LIN {X 0,Y 305.497,Z 546.552,A -85,B 0,C 180,E1 -15897.566,E2 -15897.566} C_VEL
LIN {X 0,Y 308.122,Z 558.584,A -85,B 0,C 180,E1 -15901.379,E2 -15901.379} C_VEL
LIN {X 0,Y 309.792,Z 567.618,A -85,B 0,C 180,E1 -15904.104,E2 -15904.104} C_VEL
LIN {X 0,Y 309.747,Z 569.897,A -85,B 0,C 180,E1 -15904.748,E2 -15904.748} C_VEL
LIN {X 0,Y 315.852,Z 610.316,A -85,B 0,C 180,E1 -15906.253,E2 -15906.253} C_VEL
LIN {X 0,Y 314.086,Z 678.463,A -85,B 0,C 180,E1 -15907.943,E2 -15907.943} C_VEL
LIN {X 0,Y 313.22,Z 691.999,A -85,B 0,C 180,E1 -15908.528,E2 -15908.528} C_VEL
LIN {X 0,Y 312.136,Z 704.365,A -85,B 0,C 180,E1 -15909.314,E2 -15909.314} C_VEL
LIN {X 0,Y 310.892,Z 716.286,A -85,B 0,C 180,E1 -15910.349,E2 -15910.349} C_VEL
LIN {X 0,Y 309.544,Z 727.77,A -85,B 0,C 180,E1 -15911.636,E2 -15911.636} C_VEL
LIN {X 0,Y 308.303,Z 737.547,A -85,B 0,C 180,E1 -15913.006,E2 -15913.006} C_VEL
LIN {X 0,Y 307.077,Z 747.457,A -85,B 0,C 180,E1 -15914.738,E2 -15914.738} C_VEL
LIN {X 0,Y 305.804,Z 756.501,A -85,B 0,C 180,E1 -15916.712,E2 -15916.712} C_VEL
LIN {X 0,Y 304.877,Z 763.765,A -85,B 0,C 180,E1 -15918.698,E2 -15918.698} C_VEL
LIN {X 0,Y 304.247,Z 769.534,A -85,B 0,C 180,E1 -15920.693,E2 -15920.693} C_VEL
LIN {X 0,Y 303.857,Z 774.057,A -85,B 0,C 180,E1 -15922.69,E2 -15922.69} C_VEL
LIN {X 0,Y 303.669,Z 777.467,A -85,B 0,C 180,E1 -15924.686,E2 -15924.686} C_VEL
LIN {X 0,Y 303.642,Z 779.152,A -85,B 0,C 180,E1 -15926.016,E2 -15926.016} C_VEL
LIN {X 0,Y 303.61,Z 780.42,A -85,B 0,C 180,E1 -15927.345,E2 -15927.345} C_VEL
LIN {X 0,Y 303.577,Z 781.275,A -85,B 0,C 180,E1 -15928.672,E2 -15928.672} C_VEL
LIN {X 0,Y 303.605,Z 781.68,A -85,B 0,C 180,E1 -15929.998,E2 -15929.998} C_VEL
LIN {X 0,Y 303.567,Z 781.681,A -85,B 0,C 180,E1 -15931.325,E2 -15931.325} C_VEL
LIN {X 0,Y 303.604,Z 781.289,A -85,B 0,C 180,E1 -15932.652,E2 -15932.652} C_VEL
LIN {X 0,Y 303.599,Z 780.496,A -85,B 0,C 180,E1 -15933.98,E2 -15933.98} C_VEL
LIN {X 0,Y 303.626,Z 778.989,A -85,B 0,C 180,E1 -15935.543,E2 -15935.543} C_VEL
LIN {X 0,Y 303.993,Z 775.521,A -85,B 0,C 180,E1 -15937.971,E2 -15937.971} C_VEL
LIN {X 0,Y 304.505,Z 771.506,A -85,B 0,C 180,E1 -15939.966,E2 -15939.966} C_VEL
LIN {X 0,Y 305.464,Z 765.357,A -85,B 0,C 180,E1 -15942.286,E2 -15942.286} C_VEL
LIN {X 0,Y 306.731,Z 758.652,A -85,B 0,C 180,E1 -15944.257,E2 -15944.257} C_VEL
LIN {X 0,Y 308.205,Z 750.629,A -85,B 0,C 180,E1 -15946.157,E2 -15946.157} C_VEL
LIN {X 0,Y 309.648,Z 741.904,A -85,B 0,C 180,E1 -15947.84,E2 -15947.84} C_VEL
LIN {X 0,Y 311.396,Z 731.495,A -85,B 0,C 180,E1 -15949.443,E2 -15949.443} C_VEL
LIN {X 0,Y 313.245,Z 719.826,A -85,B 0,C 180,E1 -15950.863,E2 -15950.863} C_VEL
LIN {X 0,Y 314.876,Z 708.285,A -85,B 0,C 180,E1 -15951.952,E2 -15951.952} C_VEL
LIN {X 0,Y 316.109,Z 696.459,A -85,B 0,C 180,E1 -15952.808,E2 -15952.808} C_VEL
LIN {X 0,Y 317.302,Z 683.01,A -85,B 0,C 180,E1 -15953.494,E2 -15953.494} C_VEL
LIN {X 0,Y 318.066,Z 670,A -85,B 0,C 180,E1 -15953.9,E2 -15953.9} C_VEL
LIN {X 0,Y 319.853,Z 610.651,A -85,B 0,C 180,E1 -15955.385,E2 -15955.385} C_VEL
LIN {X 0,Y 316.871,Z 591.359,A -85,B 0,C 180,E1 -15956.251,E2 -15956.251} C_VEL
LIN {X 0,Y 313.731,Z 576.118,A -85,B 0,C 180,E1 -15957.04,E2 -15957.04} C_VEL
LIN {X 0,Y 310.518,Z 568.505,A -85,B 0,C 180,E1 -15957.655,E2 -15957.655} C_VEL
LIN {X 0,Y 309.018,Z 560.982,A -85,B 0,C 180,E1 -15960.203,E2 -15960.203} C_VEL
LIN {X 0,Y 306.966,Z 552.375,A -85,B 0,C 180,E1 -15963.329,E2 -15963.329} C_VEL
LIN {X 0,Y 305.5,Z 546.432,A -85,B 0,C 180,E1 -15965.712,E2 -15965.712} C_VEL
LIN {X 0,Y 305.488,Z 546.436,A -85,B 0,C 180,E1 -15968.537,E2 -15968.537} C_VEL
LIN {X 0,Y 305.483,Z 546.436,A -85,B 0,C 180,E1 -15972.591,E2 -15972.591} C_VEL
LIN {X 0,Y 305.482,Z 546.432,A -85,B 0,C 180,E1 -15977.405,E2 -15977.405} C_VEL
LIN {X 0,Y 305.501,Z 546.43,A -85,B 0,C 180,E1 -15981.601,E2 -15981.601} C_VEL
LIN {X 0,Y 305.455,Z 546.436,A -85,B 0,C 180,E1 -15984.885,E2 -15984.885} C_VEL
LIN {X 0,Y 305.444,Z 546.435,A -85,B 0,C 180,E1 -15988.353,E2 -15988.353} C_VEL
LIN {X 0,Y 305.512,Z 546.43,A -85,B 0,C 180,E1 -15991.112,E2 -15991.112} C_VEL
LIN {X 0,Y 305.562,Z 546.423,A -85,B 0,C 180,E1 -15994.086,E2 -15994.086} C_VEL
LIN {X 0,Y 305.491,Z 546.431,A -85,B 0,C 180,E1 -15998.401,E2 -15998.401} C_VEL
LIN {X 0,Y 305.58,Z 546.413,A -85,B 0,C 180,E1 -16001.216,E2 -16001.216} C_VEL
LIN {X 0,Y 305.638,Z 546.409,A -85,B 0,C 180,E1 -16005.348,E2 -16005.348} C_VEL
LIN {X 0,Y 305.63,Z 546.412,A -85,B 0,C 180,E1 -16009.399,E2 -16009.399} C_VEL
LIN {X 0,Y 305.802,Z 546.386,A -85,B 0,C 180,E1 -16012.073,E2 -16012.073} C_VEL
LIN {X 0,Y 305.68,Z 546.405,A -85,B 0,C 180,E1 -16014.723,E2 -16014.723} C_VEL
LIN {X 0,Y 305.95,Z 546.368,A -85,B 0,C 180,E1 -16018.683,E2 -16018.683} C_VEL
LIN {X 0,Y 305.95,Z 546.372,A -85,B 0,C 180,E1 -16021.316,E2 -16021.316} C_VEL
LIN {X 0,Y 305.682,Z 546.405,A -85,B 0,C 180,E1 -16025.276,E2 -16025.276} C_VEL
LIN {X 0,Y 305.802,Z 546.392,A -85,B 0,C 180,E1 -16027.925,E2 -16027.925} C_VEL
LIN {X 0,Y 305.595,Z 546.418,A -85,B 0,C 180,E1 -16031.945,E2 -16031.945} C_VEL
LIN {X 0,Y 305.626,Z 546.419,A -85,B 0,C 180,E1 -16035.035,E2 -16035.035} C_VEL
LIN {X 0,Y 305.596,Z 546.587,A -85,B 0,C 180,E1 -16038.607,E2 -16038.607} C_VEL
LIN {X 0,Y 307.529,Z 554.976,A -85,B 0,C 180,E1 -16042.064,E2 -16042.064} C_VEL
LIN {X 0,Y 316.004,Z 572.925,A -85,B 0,C 180,E1 -16043.598,E2 -16043.598} C_VEL
LIN {X 0,Y 319.551,Z 581.78,A -85,B 0,C 180,E1 -16044.238,E2 -16044.238} C_VEL
LIN {X 0,Y 320.605,Z 586.987,A -85,B 0,C 180,E1 -16044.497,E2 -16044.497} C_VEL
LIN {X 0,Y 318.005,Z 661.781,A -85,B 0,C 180,E1 -16046.382,E2 -16046.382} C_VEL
LIN {X 0,Y 317.129,Z 675.045,A -85,B 0,C 180,E1 -16046.96,E2 -16046.96} C_VEL
LIN {X 0,Y 316.022,Z 687.675,A -85,B 0,C 180,E1 -16047.771,E2 -16047.771} C_VEL
LIN {X 0,Y 314.756,Z 698.402,A -85,B 0,C 180,E1 -16048.689,E2 -16048.689} C_VEL
LIN {X 0,Y 313.17,Z 709.886,A -85,B 0,C 180,E1 -16049.954,E2 -16049.954} C_VEL
LIN {X 0,Y 311.449,Z 720.68,A -85,B 0,C 180,E1 -16051.454,E2 -16051.454} C_VEL
LIN {X 0,Y 309.689,Z 730.59,A -85,B 0,C 180,E1 -16053.194,E2 -16053.194} C_VEL
LIN {X 0,Y 308.019,Z 739.585,A -85,B 0,C 180,E1 -16055.182,E2 -16055.182} C_VEL
LIN {X 0,Y 306.727,Z 746.339,A -85,B 0,C 180,E1 -16057.049,E2 -16057.049} C_VEL
LIN {X 0,Y 305.478,Z 752.794,A -85,B 0,C 180,E1 -16059.333,E2 -16059.333} C_VEL
LIN {X 0,Y 304.787,Z 756.885,A -85,B 0,C 180,E1 -16061.202,E2 -16061.202} C_VEL
LIN {X 0,Y 304.193,Z 760.192,A -85,B 0,C 180,E1 -16063.191,E2 -16063.191} C_VEL
LIN {X 0,Y 303.966,Z 761.501,A -85,B 0,C 180,E1 -16064.216,E2 -16064.216} C_VEL
LIN {X 0,Y 303.625,Z 763.205,A -85,B 0,C 180,E1 -16066.023,E2 -16066.023} C_VEL
LIN {X 0,Y 303.417,Z 764.115,A -85,B 0,C 180,E1 -16067.833,E2 -16067.833} C_VEL
LIN {X 0,Y 303.29,Z 764.261,A -85,B 0,C 180,E1 -16069.879,E2 -16069.879} C_VEL
LIN {X 0,Y 303.332,Z 763.417,A -85,B 0,C 180,E1 -16071.975,E2 -16071.975} C_VEL
LIN {X 0,Y 303.671,Z 760.861,A -85,B 0,C 180,E1 -16074.652,E2 -16074.652} C_VEL
LIN {X 0,Y 304.083,Z 756.872,A -85,B 0,C 180,E1 -16077.134,E2 -16077.134} C_VEL
LIN {X 0,Y 304.716,Z 751.498,A -85,B 0,C 180,E1 -16079.511,E2 -16079.511} C_VEL
LIN {X 0,Y 305.463,Z 745.633,A -85,B 0,C 180,E1 -16081.486,E2 -16081.486} C_VEL
LIN {X 0,Y 306.437,Z 738.38,A -85,B 0,C 180,E1 -16083.436,E2 -16083.436} C_VEL
LIN {X 0,Y 307.701,Z 729.421,A -85,B 0,C 180,E1 -16085.367,E2 -16085.367} C_VEL
LIN {X 0,Y 308.945,Z 719.517,A -85,B 0,C 180,E1 -16087.075,E2 -16087.075} C_VEL
LIN {X 0,Y 310.344,Z 708.853,A -85,B 0,C 180,E1 -16088.538,E2 -16088.538} C_VEL
LIN {X 0,Y 311.485,Z 698.278,A -85,B 0,C 180,E1 -16089.704,E2 -16089.704} C_VEL
LIN {X 0,Y 312.546,Z 687.241,A -85,B 0,C 180,E1 -16090.664,E2 -16090.664} C_VEL
LIN {X 0,Y 313.439,Z 674.541,A -85,B 0,C 180,E1 -16091.488,E2 -16091.488} C_VEL
LIN {X 0,Y 314.186,Z 660.798,A -85,B 0,C 180,E1 -16092.089,E2 -16092.089} C_VEL
LIN {X 0,Y 316.226,Z 584.792,A -85,B 0,C 180,E1 -16093.966,E2 -16093.966} C_VEL
LIN {X 0,Y 313.519,Z 571.685,A -85,B 0,C 180,E1 -16094.502,E2 -16094.502} C_VEL
LIN {X 0,Y 307.021,Z 553.372,A -85,B 0,C 180,E1 -16095.503,E2 -16095.503} C_VEL
LIN {X 0,Y 305.625,Z 546.415,A -85,B 0,C 180,E1 -16097.974,E2 -16097.974} C_VEL
LIN {X 0,Y 305.799,Z 546.392,A -85,B 0,C 180,E1 -16102.076,E2 -16102.076} C_VEL
LIN {X 0,Y 305.684,Z 546.411,A -85,B 0,C 180,E1 -16104.725,E2 -16104.725} C_VEL
LIN {X 0,Y 305.954,Z 546.375,A -85,B 0,C 180,E1 -16108.686,E2 -16108.686} C_VEL
LIN {X 0,Y 305.955,Z 546.373,A -85,B 0,C 180,E1 -16111.318,E2 -16111.318} C_VEL
LIN {X 0,Y 305.844,Z 546.385,A -85,B 0,C 180,E1 -16116.599,E2 -16116.599} C_VEL
LIN {X 0,Y 305.734,Z 546.402,A -85,B 0,C 180,E1 -16119.262,E2 -16119.262} C_VEL
LIN {X 0,Y 305.588,Z 546.418,A -85,B 0,C 180,E1 -16123.298,E2 -16123.298} C_VEL
LIN {X 0,Y 305.593,Z 546.416,A -85,B 0,C 180,E1 -16126.022,E2 -16126.022} C_VEL
LIN {X 0,Y 305.577,Z 546.419,A -85,B 0,C 180,E1 -16129.447,E2 -16129.447} C_VEL
LIN {X 0,Y 305.491,Z 546.428,A -85,B 0,C 180,E1 -16133.043,E2 -16133.043} C_VEL
LIN {X 0,Y 305.526,Z 546.424,A -85,B 0,C 180,E1 -16136.221,E2 -16136.221} C_VEL
LIN {X 0,Y 305.49,Z 546.433,A -85,B 0,C 180,E1 -16139.049,E2 -16139.049} C_VEL
LIN {X 0,Y 305.443,Z 546.433,A -85,B 0,C 180,E1 -16141.954,E2 -16141.954} C_VEL
LIN {X 0,Y 305.464,Z 546.436,A -85,B 0,C 180,E1 -16145.115,E2 -16145.115} C_VEL
LIN {X 0,Y 305.443,Z 546.435,A -85,B 0,C 180,E1 -16148.528,E2 -16148.528} C_VEL
LIN {X 0,Y 305.462,Z 546.431,A -85,B 0,C 180,E1 -16152.588,E2 -16152.588} C_VEL
LIN {X 0,Y 305.446,Z 546.434,A -85,B 0,C 180,E1 -16156.35,E2 -16156.35} C_VEL
LIN {X 0,Y 305.462,Z 546.431,A -85,B 0,C 180,E1 -16159.894,E2 -16159.894} C_VEL
LIN {X 0,Y 305.43,Z 546.434,A -85,B 0,C 180,E1 -16160.94,E2 -16160.94} C_VEL
LIN {X 0,Y 304.777,Z 546.52,A -85,B 0,C 180,E1 -16162.041,E2 -16162.041} C_VEL
LIN {X 0,Y 301.908,Z 546.877,A -85,B 0,C 180,E1 -16163.831,E2 -16163.831} C_VEL
LIN {X 0,Y 299.477,Z 547.181,A -85,B 0,C 180,E1 -16165.283,E2 -16165.283} C_VEL
LIN {X 0,Y 298.453,Z 547.305,A -85,B 0,C 180,E1 -16166.409,E2 -16166.409} C_VEL
LIN {X 0,Y 298.381,Z 547.315,A -85,B 0,C 180,E1 -16166.79,E2 -16166.79} C_VEL
LIN {X 0,Y 298.437,Z 547.304,A -85,B 0,C 180,E1 -16170.616,E2 -16170.616} C_VEL
LIN {X 0,Y 298.49,Z 547.303,A -85,B 0,C 180,E1 -16173.476,E2 -16173.476} C_VEL
LIN {X 0,Y 298.437,Z 547.307,A -85,B 0,C 180,E1 -16176.701,E2 -16176.701} C_VEL
LIN {X 0,Y 298.51,Z 547.296,A -85,B 0,C 180,E1 -16180.756,E2 -16180.756} C_VEL
LIN {X 0,Y 298.593,Z 547.287,A -85,B 0,C 180,E1 -16184.995,E2 -16184.995} C_VEL
LIN {X 0,Y 298.599,Z 547.288,A -85,B 0,C 180,E1 -16189.148,E2 -16189.148} C_VEL
LIN {X 0,Y 298.749,Z 547.27,A -85,B 0,C 180,E1 -16191.886,E2 -16191.886} C_VEL
LIN {X 0,Y 298.664,Z 547.277,A -85,B 0,C 180,E1 -16194.6,E2 -16194.6} C_VEL
LIN {X 0,Y 298.93,Z 547.246,A -85,B 0,C 180,E1 -16198.654,E2 -16198.654} C_VEL
LIN {X 0,Y 298.93,Z 547.247,A -85,B 0,C 180,E1 -16201.348,E2 -16201.348} C_VEL
LIN {X 0,Y 298.806,Z 547.261,A -85,B 0,C 180,E1 -16206.754,E2 -16206.754} C_VEL
LIN {X 0,Y 298.689,Z 547.278,A -85,B 0,C 180,E1 -16209.481,E2 -16209.481} C_VEL
LIN {X 0,Y 298.56,Z 547.292,A -85,B 0,C 180,E1 -16213.616,E2 -16213.616} C_VEL
LIN {X 0,Y 298.557,Z 547.295,A -85,B 0,C 180,E1 -16216.409,E2 -16216.409} C_VEL
LIN {X 0,Y 298.507,Z 547.301,A -85,B 0,C 180,E1 -16219.647,E2 -16219.647} C_VEL
LIN {X 0,Y 298.437,Z 547.303,A -85,B 0,C 180,E1 -16223.6,E2 -16223.6} C_VEL
LIN {X 0,Y 298.498,Z 547.299,A -85,B 0,C 180,E1 -16226.574,E2 -16226.574} C_VEL
LIN {X 0,Y 298.425,Z 547.31,A -85,B 0,C 180,E1 -16229.641,E2 -16229.641} C_VEL
LIN {X 0,Y 298.403,Z 547.312,A -85,B 0,C 180,E1 -16232.8,E2 -16232.8} C_VEL
LIN {X 0,Y 298.455,Z 547.307,A -85,B 0,C 180,E1 -16236.807,E2 -16236.807} C_VEL
LIN {X 0,Y 298.417,Z 547.31,A -85,B 0,C 180,E1 -16239.486,E2 -16239.486} C_VEL
LIN {X 0,Y 298.407,Z 547.312,A -85,B 0,C 180,E1 -16243.103,E2 -16243.103} C_VEL
LIN {X 0,Y 298.411,Z 547.312,A -85,B 0,C 180,E1 -16246.92,E2 -16246.92} C_VEL
LIN {X 0,Y 298.423,Z 547.31,A -85,B 0,C 180,E1 -16251.003,E2 -16251.003} C_VEL
LIN {X 0,Y 298.44,Z 547.31,A -85,B 0,C 180,E1 -16253.931,E2 -16253.931} C_VEL
LIN {X 0,Y 298.463,Z 547.398,A -85,B 0,C 180,E1 -16257.156,E2 -16257.156} C_VEL
LIN {X 0,Y 301.028,Z 559.299,A -85,B 0,C 180,E1 -16261.022,E2 -16261.022} C_VEL
LIN {X 0,Y 302.74,Z 568.34,A -85,B 0,C 180,E1 -16263.825,E2 -16263.825} C_VEL
LIN {X 0,Y 302.887,Z 569.821,A -85,B 0,C 180,E1 -16264.238,E2 -16264.238} C_VEL
LIN {X 0,Y 309.184,Z 611.129,A -85,B 0,C 180,E1 -16265.825,E2 -16265.825} C_VEL
LIN {X 0,Y 307.369,Z 678.143,A -85,B 0,C 180,E1 -16267.524,E2 -16267.524} C_VEL
LIN {X 0,Y 306.479,Z 691.706,A -85,B 0,C 180,E1 -16268.12,E2 -16268.12} C_VEL
LIN {X 0,Y 305.37,Z 704.096,A -85,B 0,C 180,E1 -16268.922,E2 -16268.922} C_VEL
LIN {X 0,Y 304.183,Z 715.241,A -85,B 0,C 180,E1 -16269.897,E2 -16269.897} C_VEL
LIN {X 0,Y 302.746,Z 726.873,A -85,B 0,C 180,E1 -16271.208,E2 -16271.208} C_VEL
LIN {X 0,Y 301.429,Z 737.048,A -85,B 0,C 180,E1 -16272.651,E2 -16272.651} C_VEL
LIN {X 0,Y 300.205,Z 746.822,A -85,B 0,C 180,E1 -16274.38,E2 -16274.38} C_VEL
LIN {X 0,Y 298.869,Z 755.94,A -85,B 0,C 180,E1 -16276.397,E2 -16276.397} C_VEL
LIN {X 0,Y 297.862,Z 763.277,A -85,B 0,C 180,E1 -16278.429,E2 -16278.429} C_VEL
LIN {X 0,Y 297.219,Z 769.12,A -85,B 0,C 180,E1 -16280.471,E2 -16280.471} C_VEL
LIN {X 0,Y 296.801,Z 773.694,A -85,B 0,C 180,E1 -16282.515,E2 -16282.515} C_VEL
LIN {X 0,Y 296.584,Z 777.148,A -85,B 0,C 180,E1 -16284.559,E2 -16284.559} C_VEL
LIN {X 0,Y 296.541,Z 778.855,A -85,B 0,C 180,E1 -16285.921,E2 -16285.921} C_VEL
LIN {X 0,Y 296.537,Z 780.145,A -85,B 0,C 180,E1 -16287.281,E2 -16287.281} C_VEL
LIN {X 0,Y 296.496,Z 781.026,A -85,B 0,C 180,E1 -16288.64,E2 -16288.64} C_VEL
LIN {X 0,Y 296.52,Z 781.463,A -85,B 0,C 180,E1 -16289.998,E2 -16289.998} C_VEL
LIN {X 0,Y 296.486,Z 781.483,A -85,B 0,C 180,E1 -16291.356,E2 -16291.356} C_VEL
LIN {X 0,Y 296.529,Z 781.11,A -85,B 0,C 180,E1 -16292.715,E2 -16292.715} C_VEL
LIN {X 0,Y 296.501,Z 780.34,A -85,B 0,C 180,E1 -16294.076,E2 -16294.076} C_VEL
LIN {X 0,Y 296.547,Z 779.05,A -85,B 0,C 180,E1 -16295.507,E2 -16295.507} C_VEL
LIN {X 0,Y 296.948,Z 775.437,A -85,B 0,C 180,E1 -16298.162,E2 -16298.162} C_VEL
LIN {X 0,Y 297.483,Z 771.472,A -85,B 0,C 180,E1 -16300.204,E2 -16300.204} C_VEL
LIN {X 0,Y 298.331,Z 766.377,A -85,B 0,C 180,E1 -16302.239,E2 -16302.239} C_VEL
LIN {X 0,Y 299.623,Z 759.996,A -85,B 0,C 180,E1 -16304.256,E2 -16304.256} C_VEL
LIN {X 0,Y 301.126,Z 752.029,A -85,B 0,C 180,E1 -16306.262,E2 -16306.262} C_VEL
LIN {X 0,Y 302.558,Z 743.939,A -85,B 0,C 180,E1 -16307.923,E2 -16307.923} C_VEL
LIN {X 0,Y 304.374,Z 734.098,A -85,B 0,C 180,E1 -16309.558,E2 -16309.558} C_VEL
LIN {X 0,Y 306.21,Z 723.166,A -85,B 0,C 180,E1 -16311.013,E2 -16311.013} C_VEL
LIN {X 0,Y 307.811,Z 712.544,A -85,B 0,C 180,E1 -16312.129,E2 -16312.129} C_VEL
LIN {X 0,Y 309.378,Z 699.909,A -85,B 0,C 180,E1 -16313.157,E2 -16313.157} C_VEL
LIN {X 0,Y 310.708,Z 687.358,A -85,B 0,C 180,E1 -16313.891,E2 -16313.891} C_VEL
LIN {X 0,Y 311.606,Z 675.051,A -85,B 0,C 180,E1 -16314.367,E2 -16314.367} C_VEL
LIN {X 0,Y 313.668,Z 611.511,A -85,B 0,C 180,E1 -16316.005,E2 -16316.005} C_VEL
LIN {X 0,Y 310.878,Z 593.293,A -85,B 0,C 180,E1 -16316.85,E2 -16316.85} C_VEL
LIN {X 0,Y 307.992,Z 579.042,A -85,B 0,C 180,E1 -16317.615,E2 -16317.615} C_VEL
LIN {X 0,Y 303.339,Z 568.181,A -85,B 0,C 180,E1 -16318.558,E2 -16318.558} C_VEL
LIN {X 0,Y 301.482,Z 559.571,A -85,B 0,C 180,E1 -16321.633,E2 -16321.633} C_VEL
LIN {X 0,Y 299.209,Z 550.256,A -85,B 0,C 180,E1 -16325.236,E2 -16325.236} C_VEL
LIN {X 0,Y 298.47,Z 547.31,A -85,B 0,C 180,E1 -16326.489,E2 -16326.489} C_VEL
LIN {X 0,Y 298.416,Z 547.321,A -85,B 0,C 180,E1 -16329.482,E2 -16329.482} C_VEL
LIN {X 0,Y 298.42,Z 547.317,A -85,B 0,C 180,E1 -16333.107,E2 -16333.107} C_VEL
LIN {X 0,Y 298.426,Z 547.311,A -85,B 0,C 180,E1 -16336.924,E2 -16336.924} C_VEL
LIN {X 0,Y 298.419,Z 547.313,A -85,B 0,C 180,E1 -16340.999,E2 -16340.999} C_VEL
LIN {X 0,Y 298.425,Z 547.313,A -85,B 0,C 180,E1 -16343.93,E2 -16343.93} C_VEL
LIN {X 0,Y 298.387,Z 547.315,A -85,B 0,C 180,E1 -16347.982,E2 -16347.982} C_VEL
LIN {X 0,Y 298.455,Z 547.304,A -85,B 0,C 180,E1 -16351.903,E2 -16351.903} C_VEL
LIN {X 0,Y 298.477,Z 547.306,A -85,B 0,C 180,E1 -16354.923,E2 -16354.923} C_VEL
LIN {X 0,Y 298.44,Z 547.306,A -85,B 0,C 180,E1 -16359.314,E2 -16359.314} C_VEL
LIN {X 0,Y 298.528,Z 547.299,A -85,B 0,C 180,E1 -16362.178,E2 -16362.178} C_VEL
LIN {X 0,Y 298.583,Z 547.285,A -85,B 0,C 180,E1 -16364.994,E2 -16364.994} C_VEL
LIN {X 0,Y 298.585,Z 547.287,A -85,B 0,C 180,E1 -16369.146,E2 -16369.146} C_VEL
LIN {X 0,Y 298.747,Z 547.264,A -85,B 0,C 180,E1 -16371.885,E2 -16371.885} C_VEL
LIN {X 0,Y 298.651,Z 547.281,A -85,B 0,C 180,E1 -16374.598,E2 -16374.598} C_VEL
LIN {X 0,Y 298.917,Z 547.244,A -85,B 0,C 180,E1 -16378.652,E2 -16378.652} C_VEL
LIN {X 0,Y 298.917,Z 547.247,A -85,B 0,C 180,E1 -16381.347,E2 -16381.347} C_VEL
LIN {X 0,Y 298.653,Z 547.281,A -85,B 0,C 180,E1 -16385.401,E2 -16385.401} C_VEL
LIN {X 0,Y 298.747,Z 547.272,A -85,B 0,C 180,E1 -16388.114,E2 -16388.114} C_VEL
LIN {X 0,Y 298.544,Z 547.297,A -85,B 0,C 180,E1 -16392.231,E2 -16392.231} C_VEL
LIN {X 0,Y 298.578,Z 547.296,A -85,B 0,C 180,E1 -16395.198,E2 -16395.198} C_VEL
LIN {X 0,Y 298.567,Z 547.486,A -85,B 0,C 180,E1 -16397.818,E2 -16397.818} C_VEL
LIN {X 0,Y 300.413,Z 555.357,A -85,B 0,C 180,E1 -16401.17,E2 -16401.17} C_VEL
LIN {X 0,Y 309.212,Z 573.343,A -85,B 0,C 180,E1 -16402.837,E2 -16402.837} C_VEL
LIN {X 0,Y 313.732,Z 584.51,A -85,B 0,C 180,E1 -16403.687,E2 -16403.687} C_VEL
LIN {X 0,Y 314.466,Z 588.825,A -85,B 0,C 180,E1 -16403.894,E2 -16403.894} C_VEL
LIN {X 0,Y 311.725,Z 662.501,A -85,B 0,C 180,E1 -16405.791,E2 -16405.791} C_VEL
LIN {X 0,Y 310.807,Z 675.754,A -85,B 0,C 180,E1 -16406.39,E2 -16406.39} C_VEL
LIN {X 0,Y 309.745,Z 686.872,A -85,B 0,C 180,E1 -16407.113,E2 -16407.113} C_VEL
LIN {X 0,Y 308.248,Z 699.293,A -85,B 0,C 180,E1 -16408.196,E2 -16408.196} C_VEL
LIN {X 0,Y 306.64,Z 710.25,A -85,B 0,C 180,E1 -16409.437,E2 -16409.437} C_VEL
LIN {X 0,Y 304.959,Z 720.372,A -85,B 0,C 180,E1 -16410.869,E2 -16410.869} C_VEL
LIN {X 0,Y 303.271,Z 729.439,A -85,B 0,C 180,E1 -16412.447,E2 -16412.447} C_VEL
LIN {X 0,Y 301.657,Z 737.84,A -85,B 0,C 180,E1 -16414.266,E2 -16414.266} C_VEL
LIN {X 0,Y 299.997,Z 745.862,A -85,B 0,C 180,E1 -16416.445,E2 -16416.445} C_VEL
LIN {X 0,Y 298.855,Z 751.374,A -85,B 0,C 180,E1 -16418.335,E2 -16418.335} C_VEL
LIN {X 0,Y 298.018,Z 755.77,A -85,B 0,C 180,E1 -16420.23,E2 -16420.23} C_VEL
LIN {X 0,Y 297.38,Z 759.187,A -85,B 0,C 180,E1 -16422.12,E2 -16422.12} C_VEL
LIN {X 0,Y 296.766,Z 762.488,A -85,B 0,C 180,E1 -16424.731,E2 -16424.731} C_VEL
LIN {X 0,Y 296.364,Z 764.196,A -85,B 0,C 180,E1 -16427.318,E2 -16427.318} C_VEL
LIN {X 0,Y 296.2,Z 764.526,A -85,B 0,C 180,E1 -16429.399,E2 -16429.399} C_VEL
LIN {X 0,Y 296.24,Z 763.637,A -85,B 0,C 180,E1 -16431.918,E2 -16431.918} C_VEL
LIN {X 0,Y 296.559,Z 761.247,A -85,B 0,C 180,E1 -16434.539,E2 -16434.539} C_VEL
LIN {X 0,Y 296.955,Z 757.442,A -85,B 0,C 180,E1 -16437.023,E2 -16437.023} C_VEL
LIN {X 0,Y 297.621,Z 752.094,A -85,B 0,C 180,E1 -16439.492,E2 -16439.492} C_VEL
LIN {X 0,Y 298.296,Z 746.927,A -85,B 0,C 180,E1 -16441.325,E2 -16441.325} C_VEL
LIN {X 0,Y 299.396,Z 739.189,A -85,B 0,C 180,E1 -16443.515,E2 -16443.515} C_VEL
LIN {X 0,Y 300.621,Z 730.596,A -85,B 0,C 180,E1 -16445.442,E2 -16445.442} C_VEL
LIN {X 0,Y 301.937,Z 720.667,A -85,B 0,C 180,E1 -16447.237,E2 -16447.237} C_VEL
LIN {X 0,Y 303.403,Z 709.804,A -85,B 0,C 180,E1 -16448.783,E2 -16448.783} C_VEL
LIN {X 0,Y 304.732,Z 697.895,A -85,B 0,C 180,E1 -16450.13,E2 -16450.13} C_VEL
LIN {X 0,Y 305.859,Z 686.282,A -85,B 0,C 180,E1 -16451.137,E2 -16451.137} C_VEL
LIN {X 0,Y 306.786,Z 672.994,A -85,B 0,C 180,E1 -16451.987,E2 -16451.987} C_VEL
LIN {X 0,Y 307.503,Z 659.831,A -85,B 0,C 180,E1 -16452.546,E2 -16452.546} C_VEL
LIN {X 0,Y 309.58,Z 585.791,A -85,B 0,C 180,E1 -16454.403,E2 -16454.403} C_VEL
LIN {X 0,Y 307.192,Z 574.139,A -85,B 0,C 180,E1 -16454.892,E2 -16454.892} C_VEL
LIN {X 0,Y 299.884,Z 553.671,A -85,B 0,C 180,E1 -16456.016,E2 -16456.016} C_VEL
LIN {X 0,Y 298.564,Z 547.295,A -85,B 0,C 180,E1 -16458.288,E2 -16458.288} C_VEL
LIN {X 0,Y 298.744,Z 547.271,A -85,B 0,C 180,E1 -16461.888,E2 -16461.888} C_VEL
LIN {X 0,Y 298.655,Z 547.286,A -85,B 0,C 180,E1 -16464.601,E2 -16464.601} C_VEL
LIN {X 0,Y 298.921,Z 547.251,A -85,B 0,C 180,E1 -16468.655,E2 -16468.655} C_VEL
LIN {X 0,Y 298.921,Z 547.249,A -85,B 0,C 180,E1 -16471.349,E2 -16471.349} C_VEL
LIN {X 0,Y 298.79,Z 547.265,A -85,B 0,C 180,E1 -16476.756,E2 -16476.756} C_VEL
LIN {X 0,Y 298.679,Z 547.279,A -85,B 0,C 180,E1 -16479.482,E2 -16479.482} C_VEL
LIN {X 0,Y 298.551,Z 547.292,A -85,B 0,C 180,E1 -16483.617,E2 -16483.617} C_VEL
LIN {X 0,Y 298.548,Z 547.294,A -85,B 0,C 180,E1 -16486.411,E2 -16486.411} C_VEL
LIN {X 0,Y 298.512,Z 547.297,A -85,B 0,C 180,E1 -16489.657,E2 -16489.657} C_VEL
LIN {X 0,Y 298.458,Z 547.303,A -85,B 0,C 180,E1 -16493.6,E2 -16493.6} C_VEL
LIN {X 0,Y 298.486,Z 547.301,A -85,B 0,C 180,E1 -16496.577,E2 -16496.577} C_VEL
LIN {X 0,Y 298.418,Z 547.312,A -85,B 0,C 180,E1 -16499.643,E2 -16499.643} C_VEL
LIN {X 0,Y 298.396,Z 547.312,A -85,B 0,C 180,E1 -16502.802,E2 -16502.802} C_VEL
LIN {X 0,Y 298.446,Z 547.308,A -85,B 0,C 180,E1 -16506.809,E2 -16506.809} C_VEL
LIN {X 0,Y 298.391,Z 547.314,A -85,B 0,C 180,E1 -16511.09,E2 -16511.09} C_VEL
LIN {X 0,Y 298.392,Z 547.316,A -85,B 0,C 180,E1 -16515.043,E2 -16515.043} C_VEL
LIN {X 0,Y 298.391,Z 547.313,A -85,B 0,C 180,E1 -16518.914,E2 -16518.914} C_VEL
LIN {X 0,Y 298.45,Z 547.307,A -85,B 0,C 180,E1 -16523.194,E2 -16523.194} C_VEL
LIN {X 0,Y 298.381,Z 547.315,A -85,B 0,C 180,E1 -16526.79,E2 -16526.79} C_VEL
LIN {X 0,Y 297.744,Z 547.397,A -85,B 0,C 180,E1 -16527.918,E2 -16527.918} C_VEL
LIN {X 0,Y 294.915,Z 547.746,A -85,B 0,C 180,E1 -16529.754,E2 -16529.754} C_VEL
LIN {X 0,Y 292.513,Z 548.044,A -85,B 0,C 180,E1 -16531.244,E2 -16531.244} C_VEL
LIN {X 0,Y 291.501,Z 548.168,A -85,B 0,C 180,E1 -16532.398,E2 -16532.398} C_VEL
LIN {X 0,Y 291.43,Z 548.177,A -85,B 0,C 180,E1 -16532.788,E2 -16532.788} C_VEL
LIN {X 0,Y 291.39,Z 548.185,A -85,B 0,C 180,E1 -16536.426,E2 -16536.426} C_VEL
LIN {X 0,Y 291.446,Z 548.177,A -85,B 0,C 180,E1 -16540.27,E2 -16540.27} C_VEL
LIN {X 0,Y 291.505,Z 548.169,A -85,B 0,C 180,E1 -16544.666,E2 -16544.666} C_VEL
LIN {X 0,Y 291.543,Z 548.166,A -85,B 0,C 180,E1 -16548.882,E2 -16548.882} C_VEL
LIN {X 0,Y 291.696,Z 548.15,A -85,B 0,C 180,E1 -16551.689,E2 -16551.689} C_VEL
LIN {X 0,Y 291.634,Z 548.152,A -85,B 0,C 180,E1 -16554.469,E2 -16554.469} C_VEL
LIN {X 0,Y 291.896,Z 548.122,A -85,B 0,C 180,E1 -16558.621,E2 -16558.621} C_VEL
LIN {X 0,Y 291.896,Z 548.123,A -85,B 0,C 180,E1 -16561.38,E2 -16561.38} C_VEL
LIN {X 0,Y 291.755,Z 548.139,A -85,B 0,C 180,E1 -16566.918,E2 -16566.918} C_VEL
LIN {X 0,Y 291.638,Z 548.158,A -85,B 0,C 180,E1 -16569.712,E2 -16569.712} C_VEL
LIN {X 0,Y 291.53,Z 548.17,A -85,B 0,C 180,E1 -16573.951,E2 -16573.951} C_VEL
LIN {X 0,Y 291.495,Z 548.173,A -85,B 0,C 180,E1 -16576.818,E2 -16576.818} C_VEL
LIN {X 0,Y 291.46,Z 548.18,A -85,B 0,C 180,E1 -16579.875,E2 -16579.875} C_VEL
LIN {X 0,Y 291.392,Z 548.181,A -85,B 0,C 180,E1 -16584.207,E2 -16584.207} C_VEL
LIN {X 0,Y 291.43,Z 548.178,A -85,B 0,C 180,E1 -16587.272,E2 -16587.272} C_VEL
LIN {X 0,Y 291.343,Z 548.194,A -85,B 0,C 180,E1 -16590.437,E2 -16590.437} C_VEL
LIN {X 0,Y 291.353,Z 548.192,A -85,B 0,C 180,E1 -16593.698,E2 -16593.698} C_VEL
LIN {X 0,Y 291.389,Z 548.186,A -85,B 0,C 180,E1 -16597.255,E2 -16597.255} C_VEL
LIN {X 0,Y 291.342,Z 548.194,A -85,B 0,C 180,E1 -16600.642,E2 -16600.642} C_VEL
LIN {X 0,Y 291.299,Z 548.199,A -85,B 0,C 180,E1 -16604.401,E2 -16604.401} C_VEL
LIN {X 0,Y 291.334,Z 548.195,A -85,B 0,C 180,E1 -16608.403,E2 -16608.403} C_VEL
LIN {X 0,Y 291.373,Z 548.188,A -85,B 0,C 180,E1 -16611.159,E2 -16611.159} C_VEL
LIN {X 0,Y 291.393,Z 548.19,A -85,B 0,C 180,E1 -16614.628,E2 -16614.628} C_VEL
LIN {X 0,Y 291.394,Z 548.199,A -85,B 0,C 180,E1 -16616.714,E2 -16616.714} C_VEL
LIN {X 0,Y 293.929,Z 559.979,A -85,B 0,C 180,E1 -16620.647,E2 -16620.647} C_VEL
LIN {X 0,Y 295.792,Z 569.637,A -85,B 0,C 180,E1 -16623.686,E2 -16623.686} C_VEL
LIN {X 0,Y 297.196,Z 576.07,A -85,B 0,C 180,E1 -16623.978,E2 -16623.978} C_VEL
LIN {X 0,Y 302.522,Z 611.974,A -85,B 0,C 180,E1 -16625.378,E2 -16625.378} C_VEL
LIN {X 0,Y 300.671,Z 677.823,A -85,B 0,C 180,E1 -16627.085,E2 -16627.085} C_VEL
LIN {X 0,Y 299.765,Z 691.415,A -85,B 0,C 180,E1 -16627.694,E2 -16627.694} C_VEL
LIN {X 0,Y 298.62,Z 703.827,A -85,B 0,C 180,E1 -16628.513,E2 -16628.513} C_VEL
LIN {X 0,Y 297.286,Z 715.782,A -85,B 0,C 180,E1 -16629.59,E2 -16629.59} C_VEL
LIN {X 0,Y 295.812,Z 727.282,A -85,B 0,C 180,E1 -16630.931,E2 -16630.931} C_VEL
LIN {X 0,Y 294.391,Z 737.896,A -85,B 0,C 180,E1 -16632.495,E2 -16632.495} C_VEL
LIN {X 0,Y 293.069,Z 747.836,A -85,B 0,C 180,E1 -16634.347,E2 -16634.347} C_VEL
LIN {X 0,Y 291.726,Z 756.754,A -85,B 0,C 180,E1 -16636.413,E2 -16636.413} C_VEL
LIN {X 0,Y 290.746,Z 763.859,A -85,B 0,C 180,E1 -16638.495,E2 -16638.495} C_VEL
LIN {X 0,Y 290.017,Z 770.35,A -85,B 0,C 180,E1 -16640.935,E2 -16640.935} C_VEL
LIN {X 0,Y 289.643,Z 774.593,A -85,B 0,C 180,E1 -16643.03,E2 -16643.03} C_VEL
LIN {X 0,Y 289.52,Z 776.827,A -85,B 0,C 180,E1 -16644.426,E2 -16644.426} C_VEL
LIN {X 0,Y 289.444,Z 778.558,A -85,B 0,C 180,E1 -16645.821,E2 -16645.821} C_VEL
LIN {X 0,Y 289.464,Z 779.87,A -85,B 0,C 180,E1 -16647.215,E2 -16647.215} C_VEL
LIN {X 0,Y 289.418,Z 780.772,A -85,B 0,C 180,E1 -16648.607,E2 -16648.607} C_VEL
LIN {X 0,Y 289.437,Z 781.247,A -85,B 0,C 180,E1 -16649.998,E2 -16649.998} C_VEL
LIN {X 0,Y 289.408,Z 781.286,A -85,B 0,C 180,E1 -16651.39,E2 -16651.39} C_VEL
LIN {X 0,Y 289.433,Z 780.932,A -85,B 0,C 180,E1 -16652.782,E2 -16652.782} C_VEL
LIN {X 0,Y 289.457,Z 779.145,A -85,B 0,C 180,E1 -16655.444,E2 -16655.444} C_VEL
LIN {X 0,Y 289.733,Z 776.466,A -85,B 0,C 180,E1 -16657.665,E2 -16657.665} C_VEL
LIN {X 0,Y 290.265,Z 772.903,A -85,B 0,C 180,E1 -16659.756,E2 -16659.756} C_VEL
LIN {X 0,Y 291.087,Z 768.245,A -85,B 0,C 180,E1 -16661.84,E2 -16661.84} C_VEL
LIN {X 0,Y 292.491,Z 761.215,A -85,B 0,C 180,E1 -16664.256,E2 -16664.256} C_VEL
LIN {X 0,Y 294.044,Z 753.629,A -85,B 0,C 180,E1 -16666.308,E2 -16666.308} C_VEL
LIN {X 0,Y 295.498,Z 745.935,A -85,B 0,C 180,E1 -16668.008,E2 -16668.008} C_VEL
LIN {X 0,Y 297.332,Z 736.629,A -85,B 0,C 180,E1 -16669.681,E2 -16669.681} C_VEL
LIN {X 0,Y 299.184,Z 726.323,A -85,B 0,C 180,E1 -16671.17,E2 -16671.17} C_VEL
LIN {X 0,Y 301.083,Z 714.956,A -85,B 0,C 180,E1 -16672.47,E2 -16672.47} C_VEL
LIN {X 0,Y 302.678,Z 703.215,A -85,B 0,C 180,E1 -16673.519,E2 -16673.519} C_VEL
LIN {X 0,Y 304.04,Z 691.152,A -85,B 0,C 180,E1 -16674.312,E2 -16674.312} C_VEL
LIN {X 0,Y 305.205,Z 677.178,A -85,B 0,C 180,E1 -16674.936,E2 -16674.936} C_VEL
LIN {X 0,Y 307.505,Z 612.31,A -85,B 0,C 180,E1 -16676.657,E2 -16676.657} C_VEL
LIN {X 0,Y 304.7,Z 593.818,A -85,B 0,C 180,E1 -16677.554,E2 -16677.554} C_VEL
LIN {X 0,Y 302.368,Z 582.16,A -85,B 0,C 180,E1 -16678.204,E2 -16678.204} C_VEL
LIN {X 0,Y 296.176,Z 567.959,A -85,B 0,C 180,E1 -16679.49,E2 -16679.49} C_VEL
LIN {X 0,Y 293.914,Z 558.181,A -85,B 0,C 180,E1 -16683.183,E2 -16683.183} C_VEL
LIN {X 0,Y 291.873,Z 549.93,A -85,B 0,C 180,E1 -16686.577,E2 -16686.577} C_VEL
LIN {X 0,Y 291.407,Z 548.189,A -85,B 0,C 180,E1 -16687.353,E2 -16687.353} C_VEL
LIN {X 0,Y 291.372,Z 548.195,A -85,B 0,C 180,E1 -16690.633,E2 -16690.633} C_VEL
LIN {X 0,Y 291.317,Z 548.2,A -85,B 0,C 180,E1 -16694.393,E2 -16694.393} C_VEL
LIN {X 0,Y 291.349,Z 548.195,A -85,B 0,C 180,E1 -16698.396,E2 -16698.396} C_VEL
LIN {X 0,Y 291.368,Z 548.192,A -85,B 0,C 180,E1 -16701.16,E2 -16701.16} C_VEL
LIN {X 0,Y 291.378,Z 548.19,A -85,B 0,C 180,E1 -16704.628,E2 -16704.628} C_VEL
LIN {X 0,Y 291.364,Z 548.19,A -85,B 0,C 180,E1 -16707.949,E2 -16707.949} C_VEL
LIN {X 0,Y 291.374,Z 548.192,A -85,B 0,C 180,E1 -16711.157,E2 -16711.157} C_VEL
LIN {X 0,Y 291.408,Z 548.186,A -85,B 0,C 180,E1 -16714.27,E2 -16714.27} C_VEL
LIN {X 0,Y 291.372,Z 548.183,A -85,B 0,C 180,E1 -16717.298,E2 -16717.298} C_VEL
LIN {X 0,Y 291.448,Z 548.17,A -85,B 0,C 180,E1 -16720.269,E2 -16720.269} C_VEL
LIN {X 0,Y 291.545,Z 548.159,A -85,B 0,C 180,E1 -16724.622,E2 -16724.622} C_VEL
LIN {X 0,Y 291.528,Z 548.164,A -85,B 0,C 180,E1 -16728.88,E2 -16728.88} C_VEL
LIN {X 0,Y 291.698,Z 548.142,A -85,B 0,C 180,E1 -16731.687,E2 -16731.687} C_VEL
LIN {X 0,Y 291.621,Z 548.158,A -85,B 0,C 180,E1 -16734.467,E2 -16734.467} C_VEL
LIN {X 0,Y 291.883,Z 548.12,A -85,B 0,C 180,E1 -16738.62,E2 -16738.62} C_VEL
LIN {X 0,Y 291.883,Z 548.123,A -85,B 0,C 180,E1 -16741.379,E2 -16741.379} C_VEL
LIN {X 0,Y 291.737,Z 548.143,A -85,B 0,C 180,E1 -16746.917,E2 -16746.917} C_VEL
LIN {X 0,Y 291.618,Z 548.157,A -85,B 0,C 180,E1 -16749.712,E2 -16749.712} C_VEL
LIN {X 0,Y 291.511,Z 548.174,A -85,B 0,C 180,E1 -16753.95,E2 -16753.95} C_VEL
LIN {X 0,Y 291.487,Z 548.276,A -85,B 0,C 180,E1 -16756.907,E2 -16756.907} C_VEL
LIN {X 0,Y 293.234,Z 555.552,A -85,B 0,C 180,E1 -16760.188,E2 -16760.188} C_VEL
LIN {X 0,Y 295.225,Z 559.396,A -85,B 0,C 180,E1 -16760.6,E2 -16760.6} C_VEL
LIN {X 0,Y 302.522,Z 574.156,A -85,B 0,C 180,E1 -16762.044,E2 -16762.044} C_VEL
LIN {X 0,Y 307.853,Z 586.807,A -85,B 0,C 180,E1 -16763.088,E2 -16763.088} C_VEL
LIN {X 0,Y 308.362,Z 589.422,A -85,B 0,C 180,E1 -16763.228,E2 -16763.228} C_VEL
LIN {X 0,Y 305.494,Z 662.973,A -85,B 0,C 180,E1 -16765.165,E2 -16765.165} C_VEL
LIN {X 0,Y 304.509,Z 676.432,A -85,B 0,C 180,E1 -16765.79,E2 -16765.79} C_VEL
LIN {X 0,Y 303.184,Z 689.442,A -85,B 0,C 180,E1 -16766.687,E2 -16766.687} C_VEL
LIN {X 0,Y 301.638,Z 701.136,A -85,B 0,C 180,E1 -16767.773,E2 -16767.773} C_VEL
LIN {X 0,Y 299.926,Z 712.2,A -85,B 0,C 180,E1 -16769.092,E2 -16769.092} C_VEL
LIN {X 0,Y 298.049,Z 722.602,A -85,B 0,C 180,E1 -16770.657,E2 -16770.657} C_VEL
LIN {X 0,Y 296.257,Z 731.491,A -85,B 0,C 180,E1 -16772.317,E2 -16772.317} C_VEL
LIN {X 0,Y 294.578,Z 739.714,A -85,B 0,C 180,E1 -16774.221,E2 -16774.221} C_VEL
LIN {X 0,Y 293.107,Z 746.473,A -85,B 0,C 180,E1 -16776.153,E2 -16776.153} C_VEL
LIN {X 0,Y 291.905,Z 751.934,A -85,B 0,C 180,E1 -16778.094,E2 -16778.094} C_VEL
LIN {X 0,Y 291.015,Z 756.278,A -85,B 0,C 180,E1 -16780.043,E2 -16780.043} C_VEL
LIN {X 0,Y 290.541,Z 758.779,A -85,B 0,C 180,E1 -16781.424,E2 -16781.424} C_VEL
LIN {X 0,Y 289.958,Z 761.483,A -85,B 0,C 180,E1 -16783.356,E2 -16783.356} C_VEL
LIN {X 0,Y 289.569,Z 763.328,A -85,B 0,C 180,E1 -16785.267,E2 -16785.267} C_VEL
LIN {X 0,Y 289.307,Z 764.404,A -85,B 0,C 180,E1 -16787.145,E2 -16787.145} C_VEL
LIN {X 0,Y 289.138,Z 764.76,A -85,B 0,C 180,E1 -16788.986,E2 -16788.986} C_VEL
LIN {X 0,Y 289.115,Z 764.281,A -85,B 0,C 180,E1 -16791.065,E2 -16791.065} C_VEL
LIN {X 0,Y 289.267,Z 762.771,A -85,B 0,C 180,E1 -16793.297,E2 -16793.297} C_VEL
LIN {X 0,Y 289.63,Z 760.101,A -85,B 0,C 180,E1 -16795.59,E2 -16795.59} C_VEL
LIN {X 0,Y 290.124,Z 755.993,A -85,B 0,C 180,E1 -16797.976,E2 -16797.976} C_VEL
LIN {X 0,Y 290.87,Z 750.198,A -85,B 0,C 180,E1 -16800.438,E2 -16800.438} C_VEL
LIN {X 0,Y 291.907,Z 742.974,A -85,B 0,C 180,E1 -16802.78,E2 -16802.78} C_VEL
LIN {X 0,Y 292.964,Z 735.475,A -85,B 0,C 180,E1 -16804.701,E2 -16804.701} C_VEL
LIN {X 0,Y 294.364,Z 726.203,A -85,B 0,C 180,E1 -16806.616,E2 -16806.616} C_VEL
LIN {X 0,Y 295.596,Z 717.028,A -85,B 0,C 180,E1 -16808.156,E2 -16808.156} C_VEL
LIN {X 0,Y 296.972,Z 706.554,A -85,B 0,C 180,E1 -16809.571,E2 -16809.571} C_VEL
LIN {X 0,Y 298.256,Z 694.785,A -85,B 0,C 180,E1 -16810.829,E2 -16810.829} C_VEL
LIN {X 0,Y 299.361,Z 683.099,A -85,B 0,C 180,E1 -16811.79,E2 -16811.79} C_VEL
LIN {X 0,Y 300.256,Z 670.233,A -85,B 0,C 180,E1 -16812.56,E2 -16812.56} C_VEL
LIN {X 0,Y 300.92,Z 656.575,A -85,B 0,C 180,E1 -16813.08,E2 -16813.08} C_VEL
LIN {X 0,Y 302.944,Z 586.646,A -85,B 0,C 180,E1 -16814.861,E2 -16814.861} C_VEL
LIN {X 0,Y 300.711,Z 576.041,A -85,B 0,C 180,E1 -16815.322,E2 -16815.322} C_VEL
LIN {X 0,Y 292.674,Z 553.867,A -85,B 0,C 180,E1 -16816.595,E2 -16816.595} C_VEL
LIN {X 0,Y 291.543,Z 548.171,A -85,B 0,C 180,E1 -16818.707,E2 -16818.707} C_VEL
LIN {X 0,Y 291.692,Z 548.15,A -85,B 0,C 180,E1 -16821.69,E2 -16821.69} C_VEL
LIN {X 0,Y 291.625,Z 548.161,A -85,B 0,C 180,E1 -16824.47,E2 -16824.47} C_VEL
LIN {X 0,Y 291.887,Z 548.127,A -85,B 0,C 180,E1 -16828.622,E2 -16828.622} C_VEL
LIN {X 0,Y 291.887,Z 548.125,A -85,B 0,C 180,E1 -16831.382,E2 -16831.382} C_VEL
LIN {X 0,Y 291.739,Z 548.144,A -85,B 0,C 180,E1 -16836.92,E2 -16836.92} C_VEL
LIN {X 0,Y 291.628,Z 548.157,A -85,B 0,C 180,E1 -16839.714,E2 -16839.714} C_VEL
LIN {X 0,Y 291.521,Z 548.167,A -85,B 0,C 180,E1 -16843.952,E2 -16843.952} C_VEL
LIN {X 0,Y 291.487,Z 548.176,A -85,B 0,C 180,E1 -16846.82,E2 -16846.82} C_VEL
LIN {X 0,Y 291.451,Z 548.175,A -85,B 0,C 180,E1 -16849.877,E2 -16849.877} C_VEL
LIN {X 0,Y 291.4,Z 548.18,A -85,B 0,C 180,E1 -16854.207,E2 -16854.207} C_VEL
LIN {X 0,Y 291.42,Z 548.187,A -85,B 0,C 180,E1 -16857.274,E2 -16857.274} C_VEL
LIN {X 0,Y 291.336,Z 548.192,A -85,B 0,C 180,E1 -16860.439,E2 -16860.439} C_VEL
LIN {X 0,Y 291.346,Z 548.192,A -85,B 0,C 180,E1 -16863.7,E2 -16863.7} C_VEL
LIN {X 0,Y 291.375,Z 548.193,A -85,B 0,C 180,E1 -16867.255,E2 -16867.255} C_VEL
LIN {X 0,Y 291.335,Z 548.19,A -85,B 0,C 180,E1 -16870.644,E2 -16870.644} C_VEL
LIN {X 0,Y 291.317,Z 548.194,A -85,B 0,C 180,E1 -16874.399,E2 -16874.399} C_VEL
LIN {X 0,Y 291.33,Z 548.191,A -85,B 0,C 180,E1 -16878.406,E2 -16878.406} C_VEL
LIN {X 0,Y 291.357,Z 548.188,A -85,B 0,C 180,E1 -16881.16,E2 -16881.16} C_VEL
LIN {X 0,Y 291.366,Z 548.188,A -85,B 0,C 180,E1 -16884.628,E2 -16884.628} C_VEL
LIN {X 0,Y 291.377,Z 548.187,A -85,B 0,C 180,E1 -16887.952,E2 -16887.952} C_VEL
LIN {X 0,Y 291.388,Z 548.184,A -85,B 0,C 180,E1 -16891.16,E2 -16891.16} C_VEL
LIN {X 0,Y 291.43,Z 548.177,A -85,B 0,C 180,E1 -16892.788,E2 -16892.788} C_VEL
LIN {X 0,Y 290.778,Z 548.263,A -85,B 0,C 180,E1 -16893.942,E2 -16893.942} C_VEL
LIN {X 0,Y 287.884,Z 548.625,A -85,B 0,C 180,E1 -16895.82,E2 -16895.82} C_VEL
LIN {X 0,Y 285.428,Z 548.931,A -85,B 0,C 180,E1 -16897.345,E2 -16897.345} C_VEL
LIN {X 0,Y 284.393,Z 549.056,A -85,B 0,C 180,E1 -16898.527,E2 -16898.527} C_VEL
LIN {X 0,Y 284.32,Z 549.063,A -85,B 0,C 180,E1 -16898.928,E2 -16898.928} C_VEL
LIN {X 0,Y 284.395,Z 549.05,A -85,B 0,C 180,E1 -16902.751,E2 -16902.751} C_VEL
LIN {X 0,Y 284.47,Z 549.05,A -85,B 0,C 180,E1 -16905.697,E2 -16905.697} C_VEL
LIN {X 0,Y 284.527,Z 549.041,A -85,B 0,C 180,E1 -16910.044,E2 -16910.044} C_VEL
LIN {X 0,Y 284.694,Z 549.015,A -85,B 0,C 180,E1 -16912.911,E2 -16912.911} C_VEL
LIN {X 0,Y 284.862,Z 548.999,A -85,B 0,C 180,E1 -16918.587,E2 -16918.587} C_VEL
LIN {X 0,Y 284.862,Z 549,A -85,B 0,C 180,E1 -16921.414,E2 -16921.414} C_VEL
LIN {X 0,Y 284.707,Z 549.018,A -85,B 0,C 180,E1 -16927.091,E2 -16927.091} C_VEL
LIN {X 0,Y 284.575,Z 549.039,A -85,B 0,C 180,E1 -16929.956,E2 -16929.956} C_VEL
LIN {X 0,Y 284.49,Z 549.047,A -85,B 0,C 180,E1 -16934.303,E2 -16934.303} C_VEL
LIN {X 0,Y 284.432,Z 549.053,A -85,B 0,C 180,E1 -16937.249,E2 -16937.249} C_VEL
LIN {X 0,Y 284.386,Z 549.058,A -85,B 0,C 180,E1 -16940.242,E2 -16940.242} C_VEL
LIN {X 0,Y 284.347,Z 549.055,A -85,B 0,C 180,E1 -16944.846,E2 -16944.846} C_VEL
LIN {X 0,Y 284.338,Z 549.066,A -85,B 0,C 180,E1 -16948.011,E2 -16948.011} C_VEL
LIN {X 0,Y 284.302,Z 549.068,A -85,B 0,C 180,E1 -16951.274,E2 -16951.274} C_VEL
LIN {X 0,Y 284.35,Z 549.063,A -85,B 0,C 180,E1 -16955.348,E2 -16955.348} C_VEL
LIN {X 0,Y 284.327,Z 549.071,A -85,B 0,C 180,E1 -16958.167,E2 -16958.167} C_VEL
LIN {X 0,Y 284.278,Z 549.076,A -85,B 0,C 180,E1 -16962.124,E2 -16962.124} C_VEL
LIN {X 0,Y 284.264,Z 549.075,A -85,B 0,C 180,E1 -16966.189,E2 -16966.189} C_VEL
LIN {X 0,Y 284.315,Z 549.069,A -85,B 0,C 180,E1 -16970.023,E2 -16970.023} C_VEL
LIN {X 0,Y 284.358,Z 549.063,A -85,B 0,C 180,E1 -16973.616,E2 -16973.616} C_VEL
LIN {X 0,Y 284.402,Z 549.217,A -85,B 0,C 180,E1 -16976.335,E2 -16976.335} C_VEL
LIN {X 0,Y 286.808,Z 560.686,A -85,B 0,C 180,E1 -16980.262,E2 -16980.262} C_VEL
LIN {X 0,Y 288.599,Z 569.511,A -85,B 0,C 180,E1 -16983.104,E2 -16983.104} C_VEL
LIN {X 0,Y 290.502,Z 576.335,A -85,B 0,C 180,E1 -16983.461,E2 -16983.461} C_VEL
LIN {X 0,Y 295.871,Z 612.462,A -85,B 0,C 180,E1 -16984.914,E2 -16984.914} C_VEL
LIN {X 0,Y 293.92,Z 678.249,A -85,B 0,C 180,E1 -16986.668,E2 -16986.668} C_VEL
LIN {X 0,Y 292.976,Z 691.623,A -85,B 0,C 180,E1 -16987.288,E2 -16987.288} C_VEL
LIN {X 0,Y 291.776,Z 704.433,A -85,B 0,C 180,E1 -16988.169,E2 -16988.169} C_VEL
LIN {X 0,Y 290.401,Z 716.193,A -85,B 0,C 180,E1 -16989.27,E2 -16989.27} C_VEL
LIN {X 0,Y 288.885,Z 727.583,A -85,B 0,C 180,E1 -16990.64,E2 -16990.64} C_VEL
LIN {X 0,Y 287.409,Z 738.272,A -85,B 0,C 180,E1 -16992.274,E2 -16992.274} C_VEL
LIN {X 0,Y 286.211,Z 747.139,A -85,B 0,C 180,E1 -16993.962,E2 -16993.962} C_VEL
LIN {X 0,Y 284.797,Z 756.143,A -85,B 0,C 180,E1 -16996.076,E2 -16996.076} C_VEL
LIN {X 0,Y 283.736,Z 763.353,A -85,B 0,C 180,E1 -16998.207,E2 -16998.207} C_VEL
LIN {X 0,Y 283.153,Z 768.229,A -85,B 0,C 180,E1 -16999.992,E2 -16999.992} C_VEL
LIN {X 0,Y 282.683,Z 772.925,A -85,B 0,C 180,E1 -17002.139,E2 -17002.139} C_VEL
LIN {X 0,Y 282.412,Z 776.797,A -85,B 0,C 180,E1 -17004.524,E2 -17004.524} C_VEL
LIN {X 0,Y 282.37,Z 779.582,A -85,B 0,C 180,E1 -17007.145,E2 -17007.145} C_VEL
LIN {X 0,Y 282.342,Z 780.507,A -85,B 0,C 180,E1 -17008.572,E2 -17008.572} C_VEL
LIN {X 0,Y 282.357,Z 781.023,A -85,B 0,C 180,E1 -17009.998,E2 -17009.998} C_VEL
LIN {X 0,Y 282.332,Z 781.09,A -85,B 0,C 180,E1 -17011.424,E2 -17011.424} C_VEL
LIN {X 0,Y 282.339,Z 780.758,A -85,B 0,C 180,E1 -17012.852,E2 -17012.852} C_VEL
LIN {X 0,Y 282.367,Z 779.185,A -85,B 0,C 180,E1 -17015.381,E2 -17015.381} C_VEL
LIN {X 0,Y 282.691,Z 776.388,A -85,B 0,C 180,E1 -17017.857,E2 -17017.857} C_VEL
LIN {X 0,Y 283.23,Z 772.865,A -85,B 0,C 180,E1 -17020.001,E2 -17020.001} C_VEL
LIN {X 0,Y 284.1,Z 768.261,A -85,B 0,C 180,E1 -17022.136,E2 -17022.136} C_VEL
LIN {X 0,Y 285.356,Z 762.452,A -85,B 0,C 180,E1 -17024.256,E2 -17024.256} C_VEL
LIN {X 0,Y 286.971,Z 755.196,A -85,B 0,C 180,E1 -17026.356,E2 -17026.356} C_VEL
LIN {X 0,Y 288.75,Z 746.221,A -85,B 0,C 180,E1 -17028.444,E2 -17028.444} C_VEL
LIN {X 0,Y 290.686,Z 737.035,A -85,B 0,C 180,E1 -17030.151,E2 -17030.151} C_VEL
LIN {X 0,Y 292.607,Z 726.884,A -85,B 0,C 180,E1 -17031.669,E2 -17031.669} C_VEL
LIN {X 0,Y 294.561,Z 715.686,A -85,B 0,C 180,E1 -17032.995,E2 -17032.995} C_VEL
LIN {X 0,Y 296.377,Z 703.209,A -85,B 0,C 180,E1 -17034.143,E2 -17034.143} C_VEL
LIN {X 0,Y 297.859,Z 690.518,A -85,B 0,C 180,E1 -17034.99,E2 -17034.99} C_VEL
LIN {X 0,Y 299.005,Z 677.451,A -85,B 0,C 180,E1 -17035.586,E2 -17035.586} C_VEL
LIN {X 0,Y 301.505,Z 615.332,A -85,B 0,C 180,E1 -17037.265,E2 -17037.265} C_VEL
LIN {X 0,Y 300.685,Z 607.279,A -85,B 0,C 180,E1 -17037.618,E2 -17037.618} C_VEL
LIN {X 0,Y 297.199,Z 586.803,A -85,B 0,C 180,E1 -17038.712,E2 -17038.712} C_VEL
LIN {X 0,Y 295.694,Z 582.627,A -85,B 0,C 180,E1 -17039.047,E2 -17039.047} C_VEL
LIN {X 0,Y 290.526,Z 571.282,A -85,B 0,C 180,E1 -17040.147,E2 -17040.147} C_VEL
LIN {X 0,Y 288.893,Z 567.683,A -85,B 0,C 180,E1 -17040.536,E2 -17040.536} C_VEL
LIN {X 0,Y 286.73,Z 558.148,A -85,B 0,C 180,E1 -17044.313,E2 -17044.313} C_VEL
LIN {X 0,Y 285.004,Z 551.571,A -85,B 0,C 180,E1 -17047.165,E2 -17047.165} C_VEL
LIN {X 0,Y 284.336,Z 549.071,A -85,B 0,C 180,E1 -17048.388,E2 -17048.388} C_VEL
LIN {X 0,Y 284.294,Z 549.077,A -85,B 0,C 180,E1 -17052.129,E2 -17052.129} C_VEL
LIN {X 0,Y 284.28,Z 549.078,A -85,B 0,C 180,E1 -17056.193,E2 -17056.193} C_VEL
LIN {X 0,Y 284.345,Z 549.062,A -85,B 0,C 180,E1 -17060.011,E2 -17060.011} C_VEL
LIN {X 0,Y 284.345,Z 549.064,A -85,B 0,C 180,E1 -17063.615,E2 -17063.615} C_VEL
LIN {X 0,Y 284.3,Z 549.071,A -85,B 0,C 180,E1 -17067.188,E2 -17067.188} C_VEL
LIN {X 0,Y 284.35,Z 549.064,A -85,B 0,C 180,E1 -17070.374,E2 -17070.374} C_VEL
LIN {X 0,Y 284.369,Z 549.057,A -85,B 0,C 180,E1 -17073.585,E2 -17073.585} C_VEL
LIN {X 0,Y 284.357,Z 549.054,A -85,B 0,C 180,E1 -17076.705,E2 -17076.705} C_VEL
LIN {X 0,Y 284.394,Z 549.052,A -85,B 0,C 180,E1 -17081.26,E2 -17081.26} C_VEL
LIN {X 0,Y 284.482,Z 549.038,A -85,B 0,C 180,E1 -17084.458,E2 -17084.458} C_VEL
LIN {X 0,Y 284.479,Z 549.041,A -85,B 0,C 180,E1 -17088.6,E2 -17088.6} C_VEL
LIN {X 0,Y 284.648,Z 549.021,A -85,B 0,C 180,E1 -17091.48,E2 -17091.48} C_VEL
LIN {X 0,Y 284.592,Z 549.033,A -85,B 0,C 180,E1 -17094.33,E2 -17094.33} C_VEL
LIN {X 0,Y 284.849,Z 548.996,A -85,B 0,C 180,E1 -17098.585,E2 -17098.585} C_VEL
LIN {X 0,Y 284.849,Z 548.999,A -85,B 0,C 180,E1 -17101.413,E2 -17101.413} C_VEL
LIN {X 0,Y 284.688,Z 549.02,A -85,B 0,C 180,E1 -17107.09,E2 -17107.09} C_VEL
LIN {X 0,Y 284.555,Z 549.037,A -85,B 0,C 180,E1 -17109.955,E2 -17109.955} C_VEL
LIN {X 0,Y 284.471,Z 549.053,A -85,B 0,C 180,E1 -17114.303,E2 -17114.303} C_VEL
LIN {X 0,Y 284.483,Z 549.114,A -85,B 0,C 180,E1 -17115.951,E2 -17115.951} C_VEL
LIN {X 0,Y 286.138,Z 555.8,A -85,B 0,C 180,E1 -17119.131,E2 -17119.131} C_VEL
LIN {X 0,Y 288.178,Z 559.736,A -85,B 0,C 180,E1 -17119.592,E2 -17119.592} C_VEL
LIN {X 0,Y 295.332,Z 573.785,A -85,B 0,C 180,E1 -17121.095,E2 -17121.095} C_VEL
LIN {X 0,Y 301.533,Z 587.914,A -85,B 0,C 180,E1 -17122.355,E2 -17122.355} C_VEL
LIN {X 0,Y 302.373,Z 590.825,A -85,B 0,C 180,E1 -17122.551,E2 -17122.551} C_VEL
LIN {X 0,Y 299.372,Z 662.86,A -85,B 0,C 180,E1 -17124.485,E2 -17124.485} C_VEL
LIN {X 0,Y 298.418,Z 675.64,A -85,B 0,C 180,E1 -17125.081,E2 -17125.081} C_VEL
LIN {X 0,Y 297.257,Z 686.708,A -85,B 0,C 180,E1 -17125.817,E2 -17125.817} C_VEL
LIN {X 0,Y 295.744,Z 698.34,A -85,B 0,C 180,E1 -17126.84,E2 -17126.84} C_VEL
LIN {X 0,Y 293.963,Z 709.754,A -85,B 0,C 180,E1 -17128.149,E2 -17128.149} C_VEL
LIN {X 0,Y 291.956,Z 720.743,A -85,B 0,C 180,E1 -17129.749,E2 -17129.749} C_VEL
LIN {X 0,Y 290.081,Z 729.814,A -85,B 0,C 180,E1 -17131.391,E2 -17131.391} C_VEL
LIN {X 0,Y 288.425,Z 737.456,A -85,B 0,C 180,E1 -17133.093,E2 -17133.093} C_VEL
LIN {X 0,Y 286.838,Z 744.568,A -85,B 0,C 180,E1 -17135.038,E2 -17135.038} C_VEL
LIN {X 0,Y 285.2,Z 751.505,A -85,B 0,C 180,E1 -17137.445,E2 -17137.445} C_VEL
LIN {X 0,Y 283.99,Z 756.904,A -85,B 0,C 180,E1 -17139.904,E2 -17139.904} C_VEL
LIN {X 0,Y 283.254,Z 760.394,A -85,B 0,C 180,E1 -17142.059,E2 -17142.059} C_VEL
LIN {X 0,Y 282.701,Z 762.757,A -85,B 0,C 180,E1 -17144.113,E2 -17144.113} C_VEL
LIN {X 0,Y 282.309,Z 764.278,A -85,B 0,C 180,E1 -17146.214,E2 -17146.214} C_VEL
LIN {X 0,Y 282.063,Z 764.927,A -85,B 0,C 180,E1 -17148.372,E2 -17148.372} C_VEL
LIN {X 0,Y 282.026,Z 764.638,A -85,B 0,C 180,E1 -17150.579,E2 -17150.579} C_VEL
LIN {X 0,Y 282.174,Z 762.964,A -85,B 0,C 180,E1 -17153.293,E2 -17153.293} C_VEL
LIN {X 0,Y 282.594,Z 759.711,A -85,B 0,C 180,E1 -17156.025,E2 -17156.025} C_VEL
LIN {X 0,Y 283.163,Z 755.139,A -85,B 0,C 180,E1 -17158.589,E2 -17158.589} C_VEL
LIN {X 0,Y 284.024,Z 748.878,A -85,B 0,C 180,E1 -17161.153,E2 -17161.153} C_VEL
LIN {X 0,Y 284.997,Z 742.48,A -85,B 0,C 180,E1 -17163.186,E2 -17163.186} C_VEL
LIN {X 0,Y 286.278,Z 734.04,A -85,B 0,C 180,E1 -17165.336,E2 -17165.336} C_VEL
LIN {X 0,Y 287.673,Z 724.661,A -85,B 0,C 180,E1 -17167.241,E2 -17167.241} C_VEL
LIN {X 0,Y 289.067,Z 715.12,A -85,B 0,C 180,E1 -17168.801,E2 -17168.801} C_VEL
LIN {X 0,Y 290.404,Z 704.574,A -85,B 0,C 180,E1 -17170.198,E2 -17170.198} C_VEL
LIN {X 0,Y 291.762,Z 692.249,A -85,B 0,C 180,E1 -17171.481,E2 -17171.481} C_VEL
LIN {X 0,Y 292.886,Z 680.05,A -85,B 0,C 180,E1 -17172.427,E2 -17172.427} C_VEL
LIN {X 0,Y 293.759,Z 667.453,A -85,B 0,C 180,E1 -17173.129,E2 -17173.129} C_VEL
LIN {X 0,Y 294.32,Z 655.214,A -85,B 0,C 180,E1 -17173.566,E2 -17173.566} C_VEL
LIN {X 0,Y 296.342,Z 587.794,A -85,B 0,C 180,E1 -17175.32,E2 -17175.32} C_VEL
LIN {X 0,Y 294.335,Z 578.219,A -85,B 0,C 180,E1 -17175.749,E2 -17175.749} C_VEL
LIN {X 0,Y 286.329,Z 556.477,A -85,B 0,C 180,E1 -17177.037,E2 -17177.037} C_VEL
LIN {X 0,Y 285.5,Z 554.025,A -85,B 0,C 180,E1 -17177.202,E2 -17177.202} C_VEL
LIN {X 0,Y 284.519,Z 549.044,A -85,B 0,C 180,E1 -17179.146,E2 -17179.146} C_VEL
LIN {X 0,Y 284.643,Z 549.029,A -85,B 0,C 180,E1 -17181.483,E2 -17181.483} C_VEL
LIN {X 0,Y 284.595,Z 549.036,A -85,B 0,C 180,E1 -17184.333,E2 -17184.333} C_VEL
LIN {X 0,Y 284.853,Z 549.003,A -85,B 0,C 180,E1 -17188.588,E2 -17188.588} C_VEL
LIN {X 0,Y 284.853,Z 549.001,A -85,B 0,C 180,E1 -17191.416,E2 -17191.416} C_VEL
LIN {X 0,Y 284.692,Z 549.024,A -85,B 0,C 180,E1 -17197.092,E2 -17197.092} C_VEL
LIN {X 0,Y 284.565,Z 549.036,A -85,B 0,C 180,E1 -17199.957,E2 -17199.957} C_VEL
LIN {X 0,Y 284.481,Z 549.044,A -85,B 0,C 180,E1 -17204.305,E2 -17204.305} C_VEL
LIN {X 0,Y 284.425,Z 549.057,A -85,B 0,C 180,E1 -17207.25,E2 -17207.25} C_VEL
LIN {X 0,Y 284.379,Z 549.056,A -85,B 0,C 180,E1 -17210.244,E2 -17210.244} C_VEL
LIN {X 0,Y 284.369,Z 549.056,A -85,B 0,C 180,E1 -17213.877,E2 -17213.877} C_VEL
LIN {X 0,Y 284.395,Z 549.061,A -85,B 0,C 180,E1 -17217.174,E2 -17217.174} C_VEL
LIN {X 0,Y 284.295,Z 549.071,A -85,B 0,C 180,E1 -17221.276,E2 -17221.276} C_VEL
LIN {X 0,Y 284.343,Z 549.069,A -85,B 0,C 180,E1 -17225.35,E2 -17225.35} C_VEL
LIN {X 0,Y 284.311,Z 549.067,A -85,B 0,C 180,E1 -17228.171,E2 -17228.171} C_VEL
LIN {X 0,Y 284.272,Z 549.07,A -85,B 0,C 180,E1 -17232.126,E2 -17232.126} C_VEL
LIN {X 0,Y 284.272,Z 549.072,A -85,B 0,C 180,E1 -17236.194,E2 -17236.194} C_VEL
LIN {X 0,Y 284.311,Z 549.063,A -85,B 0,C 180,E1 -17240.026,E2 -17240.026} C_VEL
LIN {X 0,Y 284.337,Z 549.068,A -85,B 0,C 180,E1 -17243.616,E2 -17243.616} C_VEL
LIN {X 0,Y 284.313,Z 549.069,A -85,B 0,C 180,E1 -17247.191,E2 -17247.191} C_VEL
LIN {X 0,Y 284.364,Z 549.056,A -85,B 0,C 180,E1 -17250.378,E2 -17250.378} C_VEL
LIN {X 0,Y 284.384,Z 549.06,A -85,B 0,C 180,E1 -17253.588,E2 -17253.588} C_VEL
LIN {X 0,Y 284.339,Z 549.063,A -85,B 0,C 180,E1 -17256.705,E2 -17256.705} C_VEL
LIN {X 0,Y 284.32,Z 549.063,A -85,B 0,C 180,E1 -17258.928,E2 -17258.928} C_VEL
LIN {X 0,Y 283.688,Z 549.144,A -85,B 0,C 180,E1 -17260.11,E2 -17260.11} C_VEL
LIN {X 0,Y 280.874,Z 549.491,A -85,B 0,C 180,E1 -17262.037,E2 -17262.037} C_VEL
LIN {X 0,Y 278.484,Z 549.791,A -85,B 0,C 180,E1 -17263.601,E2 -17263.601} C_VEL
LIN {X 0,Y 277.482,Z 549.915,A -85,B 0,C 180,E1 -17264.813,E2 -17264.813} C_VEL
LIN {X 0,Y 277.413,Z 549.925,A -85,B 0,C 180,E1 -17265.224,E2 -17265.224} C_VEL
LIN {X 0,Y 277.469,Z 549.923,A -85,B 0,C 180,E1 -17269.788,E2 -17269.788} C_VEL
LIN {X 0,Y 277.648,Z 549.892,A -85,B 0,C 180,E1 -17272.73,E2 -17272.73} C_VEL
LIN {X 0,Y 277.828,Z 549.875,A -85,B 0,C 180,E1 -17278.551,E2 -17278.551} C_VEL
LIN {X 0,Y 277.828,Z 549.876,A -85,B 0,C 180,E1 -17281.45,E2 -17281.45} C_VEL
LIN {X 0,Y 277.662,Z 549.896,A -85,B 0,C 180,E1 -17287.271,E2 -17287.271} C_VEL
LIN {X 0,Y 277.516,Z 549.915,A -85,B 0,C 180,E1 -17290.212,E2 -17290.212} C_VEL
LIN {X 0,Y 277.443,Z 549.923,A -85,B 0,C 180,E1 -17294.674,E2 -17294.674} C_VEL
LIN {X 0,Y 277.351,Z 549.934,A -85,B 0,C 180,E1 -17299.234,E2 -17299.234} C_VEL
LIN {X 0,Y 277.301,Z 549.932,A -85,B 0,C 180,E1 -17304.158,E2 -17304.158} C_VEL
LIN {X 0,Y 277.333,Z 549.934,A -85,B 0,C 180,E1 -17307.504,E2 -17307.504} C_VEL
LIN {X 0,Y 277.281,Z 549.945,A -85,B 0,C 180,E1 -17310.481,E2 -17310.481} C_VEL
LIN {X 0,Y 277.256,Z 549.949,A -85,B 0,C 180,E1 -17313.895,E2 -17313.895} C_VEL
LIN {X 0,Y 277.28,Z 549.944,A -85,B 0,C 180,E1 -17317.468,E2 -17317.468} C_VEL
LIN {X 0,Y 277.218,Z 549.951,A -85,B 0,C 180,E1 -17321.236,E2 -17321.236} C_VEL
LIN {X 0,Y 277.209,Z 549.95,A -85,B 0,C 180,E1 -17325.226,E2 -17325.226} C_VEL
LIN {X 0,Y 277.231,Z 549.949,A -85,B 0,C 180,E1 -17329.511,E2 -17329.511} C_VEL
LIN {X 0,Y 277.29,Z 549.947,A -85,B 0,C 180,E1 -17332.532,E2 -17332.532} C_VEL
LIN {X 0,Y 277.377,Z 550.112,A -85,B 0,C 180,E1 -17335.901,E2 -17335.901} C_VEL
LIN {X 0,Y 279.698,Z 561.274,A -85,B 0,C 180,E1 -17339.83,E2 -17339.83} C_VEL
LIN {X 0,Y 281.332,Z 569.064,A -85,B 0,C 180,E1 -17342.461,E2 -17342.461} C_VEL
LIN {X 0,Y 284.029,Z 577.924,A -85,B 0,C 180,E1 -17342.973,E2 -17342.973} C_VEL
LIN {X 0,Y 289.208,Z 613.567,A -85,B 0,C 180,E1 -17344.448,E2 -17344.448} C_VEL
LIN {X 0,Y 287.255,Z 677.531,A -85,B 0,C 180,E1 -17346.189,E2 -17346.189} C_VEL
LIN {X 0,Y 286.293,Z 691.06,A -85,B 0,C 180,E1 -17346.823,E2 -17346.823} C_VEL
LIN {X 0,Y 285.041,Z 703.981,A -85,B 0,C 180,E1 -17347.721,E2 -17347.721} C_VEL
LIN {X 0,Y 283.524,Z 716.588,A -85,B 0,C 180,E1 -17348.933,E2 -17348.933} C_VEL
LIN {X 0,Y 281.965,Z 727.872,A -85,B 0,C 180,E1 -17350.335,E2 -17350.335} C_VEL
LIN {X 0,Y 280.494,Z 738.047,A -85,B 0,C 180,E1 -17351.935,E2 -17351.935} C_VEL
LIN {X 0,Y 279.076,Z 748.079,A -85,B 0,C 180,E1 -17353.916,E2 -17353.916} C_VEL
LIN {X 0,Y 277.656,Z 756.868,A -85,B 0,C 180,E1 -17356.084,E2 -17356.084} C_VEL
LIN {X 0,Y 276.597,Z 763.864,A -85,B 0,C 180,E1 -17358.27,E2 -17358.27} C_VEL
LIN {X 0,Y 275.931,Z 769.455,A -85,B 0,C 180,E1 -17360.468,E2 -17360.468} C_VEL
LIN {X 0,Y 275.51,Z 773.813,A -85,B 0,C 180,E1 -17362.67,E2 -17362.67} C_VEL
LIN {X 0,Y 275.322,Z 776.711,A -85,B 0,C 180,E1 -17364.588,E2 -17364.588} C_VEL
LIN {X 0,Y 275.278,Z 779.292,A -85,B 0,C 180,E1 -17367.071,E2 -17367.071} C_VEL
LIN {X 0,Y 275.267,Z 780.242,A -85,B 0,C 180,E1 -17368.535,E2 -17368.535} C_VEL
LIN {X 0,Y 275.279,Z 780.79,A -85,B 0,C 180,E1 -17369.998,E2 -17369.998} C_VEL
LIN {X 0,Y 275.257,Z 780.895,A -85,B 0,C 180,E1 -17371.461,E2 -17371.461} C_VEL
LIN {X 0,Y 275.248,Z 780.584,A -85,B 0,C 180,E1 -17372.925,E2 -17372.925} C_VEL
LIN {X 0,Y 275.301,Z 778.78,A -85,B 0,C 180,E1 -17375.859,E2 -17375.859} C_VEL
LIN {X 0,Y 275.498,Z 777.235,A -85,B 0,C 180,E1 -17377.326,E2 -17377.326} C_VEL
LIN {X 0,Y 275.998,Z 774.121,A -85,B 0,C 180,E1 -17379.525,E2 -17379.525} C_VEL
LIN {X 0,Y 276.808,Z 769.953,A -85,B 0,C 180,E1 -17381.717,E2 -17381.717} C_VEL
LIN {X 0,Y 278.19,Z 763.595,A -85,B 0,C 180,E1 -17384.257,E2 -17384.257} C_VEL
LIN {X 0,Y 279.878,Z 756.697,A -85,B 0,C 180,E1 -17386.407,E2 -17386.407} C_VEL
LIN {X 0,Y 281.663,Z 748.239,A -85,B 0,C 180,E1 -17388.526,E2 -17388.526} C_VEL
LIN {X 0,Y 283.597,Z 739.376,A -85,B 0,C 180,E1 -17390.298,E2 -17390.298} C_VEL
LIN {X 0,Y 285.838,Z 728.659,A -85,B 0,C 180,E1 -17392.019,E2 -17392.019} C_VEL
LIN {X 0,Y 287.79,Z 718.058,A -85,B 0,C 180,E1 -17393.378,E2 -17393.378} C_VEL
LIN {X 0,Y 289.7,Z 706.288,A -85,B 0,C 180,E1 -17394.545,E2 -17394.545} C_VEL
LIN {X 0,Y 291.307,Z 694.227,A -85,B 0,C 180,E1 -17395.449,E2 -17395.449} C_VEL
LIN {X 0,Y 292.585,Z 681.297,A -85,B 0,C 180,E1 -17396.141,E2 -17396.141} C_VEL
LIN {X 0,Y 293.41,Z 667.662,A -85,B 0,C 180,E1 -17396.589,E2 -17396.589} C_VEL
LIN {X 0,Y 295.444,Z 614.163,A -85,B 0,C 180,E1 -17398.05,E2 -17398.05} C_VEL
LIN {X 0,Y 292.95,Z 597.248,A -85,B 0,C 180,E1 -17398.93,E2 -17398.93} C_VEL
LIN {X 0,Y 291.018,Z 587.469,A -85,B 0,C 180,E1 -17399.527,E2 -17399.527} C_VEL
LIN {X 0,Y 285.344,Z 575.018,A -85,B 0,C 180,E1 -17400.781,E2 -17400.781} C_VEL
LIN {X 0,Y 281.67,Z 567.394,A -85,B 0,C 180,E1 -17401.654,E2 -17401.654} C_VEL
LIN {X 0,Y 279.608,Z 558.636,A -85,B 0,C 180,E1 -17405.315,E2 -17405.315} C_VEL
LIN {X 0,Y 277.869,Z 551.986,A -85,B 0,C 180,E1 -17408.365,E2 -17408.365} C_VEL
LIN {X 0,Y 277.293,Z 549.952,A -85,B 0,C 180,E1 -17409.425,E2 -17409.425} C_VEL
LIN {X 0,Y 277.229,Z 549.958,A -85,B 0,C 180,E1 -17413.191,E2 -17413.191} C_VEL
LIN {X 0,Y 277.234,Z 549.95,A -85,B 0,C 180,E1 -17417.317,E2 -17417.317} C_VEL
LIN {X 0,Y 277.259,Z 549.947,A -85,B 0,C 180,E1 -17420.675,E2 -17420.675} C_VEL
LIN {X 0,Y 277.297,Z 549.944,A -85,B 0,C 180,E1 -17424.342,E2 -17424.342} C_VEL
LIN {X 0,Y 277.237,Z 549.951,A -85,B 0,C 180,E1 -17427.835,E2 -17427.835} C_VEL
LIN {X 0,Y 277.281,Z 549.947,A -85,B 0,C 180,E1 -17431.211,E2 -17431.211} C_VEL
LIN {X 0,Y 277.305,Z 549.943,A -85,B 0,C 180,E1 -17434.478,E2 -17434.478} C_VEL
LIN {X 0,Y 277.276,Z 549.942,A -85,B 0,C 180,E1 -17437.653,E2 -17437.653} C_VEL
LIN {X 0,Y 277.335,Z 549.928,A -85,B 0,C 180,E1 -17440.765,E2 -17440.765} C_VEL
LIN {X 0,Y 277.425,Z 549.922,A -85,B 0,C 180,E1 -17445.325,E2 -17445.325} C_VEL
LIN {X 0,Y 277.497,Z 549.921,A -85,B 0,C 180,E1 -17449.788,E2 -17449.788} C_VEL
LIN {X 0,Y 277.642,Z 549.896,A -85,B 0,C 180,E1 -17452.728,E2 -17452.728} C_VEL
LIN {X 0,Y 277.814,Z 549.873,A -85,B 0,C 180,E1 -17458.55,E2 -17458.55} C_VEL
LIN {X 0,Y 277.815,Z 549.875,A -85,B 0,C 180,E1 -17461.449,E2 -17461.449} C_VEL
LIN {X 0,Y 277.643,Z 549.897,A -85,B 0,C 180,E1 -17467.27,E2 -17467.27} C_VEL
LIN {X 0,Y 277.496,Z 549.917,A -85,B 0,C 180,E1 -17470.211,E2 -17470.211} C_VEL
LIN {X 0,Y 277.458,Z 550.125,A -85,B 0,C 180,E1 -17474.985,E2 -17474.985} C_VEL
LIN {X 0,Y 279.059,Z 556.289,A -85,B 0,C 180,E1 -17478.016,E2 -17478.016} C_VEL
LIN {X 0,Y 281.299,Z 560.294,A -85,B 0,C 180,E1 -17478.536,E2 -17478.536} C_VEL
LIN {X 0,Y 289.007,Z 575.066,A -85,B 0,C 180,E1 -17480.247,E2 -17480.247} C_VEL
LIN {X 0,Y 295.756,Z 590.457,A -85,B 0,C 180,E1 -17481.703,E2 -17481.703} C_VEL
LIN {X 0,Y 296.378,Z 592.136,A -85,B 0,C 180,E1 -17481.838,E2 -17481.838} C_VEL
LIN {X 0,Y 293.308,Z 662.961,A -85,B 0,C 180,E1 -17483.778,E2 -17483.778} C_VEL
LIN {X 0,Y 292.305,Z 675.621,A -85,B 0,C 180,E1 -17484.372,E2 -17484.372} C_VEL
LIN {X 0,Y 290.99,Z 687.679,A -85,B 0,C 180,E1 -17485.192,E2 -17485.192} C_VEL
LIN {X 0,Y 289.475,Z 698.597,A -85,B 0,C 180,E1 -17486.179,E2 -17486.179} C_VEL
LIN {X 0,Y 287.632,Z 709.701,A -85,B 0,C 180,E1 -17487.474,E2 -17487.474} C_VEL
LIN {X 0,Y 285.511,Z 720.951,A -85,B 0,C 180,E1 -17489.148,E2 -17489.148} C_VEL
LIN {X 0,Y 283.653,Z 729.448,A -85,B 0,C 180,E1 -17490.713,E2 -17490.713} C_VEL
LIN {X 0,Y 281.665,Z 738.172,A -85,B 0,C 180,E1 -17492.694,E2 -17492.694} C_VEL
LIN {X 0,Y 279.977,Z 745.239,A -85,B 0,C 180,E1 -17494.699,E2 -17494.699} C_VEL
LIN {X 0,Y 278.527,Z 751.013,A -85,B 0,C 180,E1 -17496.727,E2 -17496.727} C_VEL
LIN {X 0,Y 277.142,Z 756.758,A -85,B 0,C 180,E1 -17499.343,E2 -17499.343} C_VEL
LIN {X 0,Y 276.383,Z 760.097,A -85,B 0,C 180,E1 -17501.386,E2 -17501.386} C_VEL
LIN {X 0,Y 275.763,Z 762.61,A -85,B 0,C 180,E1 -17503.48,E2 -17503.48} C_VEL
LIN {X 0,Y 275.179,Z 764.698,A -85,B 0,C 180,E1 -17506.407,E2 -17506.407} C_VEL
LIN {X 0,Y 274.979,Z 765.149,A -85,B 0,C 180,E1 -17508.358,E2 -17508.358} C_VEL
LIN {X 0,Y 274.946,Z 764.919,A -85,B 0,C 180,E1 -17510.283,E2 -17510.283} C_VEL
LIN {X 0,Y 274.985,Z 763.869,A -85,B 0,C 180,E1 -17512.399,E2 -17512.399} C_VEL
LIN {X 0,Y 275.276,Z 761.621,A -85,B 0,C 180,E1 -17514.782,E2 -17514.782} C_VEL
LIN {X 0,Y 275.732,Z 758.047,A -85,B 0,C 180,E1 -17517.257,E2 -17517.257} C_VEL
LIN {X 0,Y 276.427,Z 752.908,A -85,B 0,C 180,E1 -17519.816,E2 -17519.816} C_VEL
LIN {X 0,Y 277.206,Z 747.593,A -85,B 0,C 180,E1 -17521.855,E2 -17521.855} C_VEL
LIN {X 0,Y 278.405,Z 739.935,A -85,B 0,C 180,E1 -17524.188,E2 -17524.188} C_VEL
LIN {X 0,Y 279.804,Z 731.122,A -85,B 0,C 180,E1 -17526.307,E2 -17526.307} C_VEL
LIN {X 0,Y 281.255,Z 721.428,A -85,B 0,C 180,E1 -17528.182,E2 -17528.182} C_VEL
LIN {X 0,Y 282.888,Z 710.405,A -85,B 0,C 180,E1 -17529.862,E2 -17529.862} C_VEL
LIN {X 0,Y 284.286,Z 698.909,A -85,B 0,C 180,E1 -17531.256,E2 -17531.256} C_VEL
LIN {X 0,Y 285.552,Z 687.056,A -85,B 0,C 180,E1 -17532.362,E2 -17532.362} C_VEL
LIN {X 0,Y 286.59,Z 674.05,A -85,B 0,C 180,E1 -17533.255,E2 -17533.255} C_VEL
LIN {X 0,Y 287.376,Z 661.225,A -85,B 0,C 180,E1 -17533.85,E2 -17533.85} C_VEL
LIN {X 0,Y 289.611,Z 588.184,A -85,B 0,C 180,E1 -17535.83,E2 -17535.83} C_VEL
LIN {X 0,Y 287.975,Z 580.535,A -85,B 0,C 180,E1 -17536.187,E2 -17536.187} C_VEL
LIN {X 0,Y 280.132,Z 559.197,A -85,B 0,C 180,E1 -17537.485,E2 -17537.485} C_VEL
LIN {X 0,Y 278.3,Z 554.168,A -85,B 0,C 180,E1 -17537.848,E2 -17537.848} C_VEL
LIN {X 0,Y 277.473,Z 549.922,A -85,B 0,C 180,E1 -17539.513,E2 -17539.513} C_VEL
LIN {X 0,Y 277.641,Z 549.903,A -85,B 0,C 180,E1 -17542.731,E2 -17542.731} C_VEL
LIN {X 0,Y 277.819,Z 549.879,A -85,B 0,C 180,E1 -17548.553,E2 -17548.553} C_VEL
LIN {X 0,Y 277.819,Z 549.877,A -85,B 0,C 180,E1 -17551.452,E2 -17551.452} C_VEL
LIN {X 0,Y 277.647,Z 549.901,A -85,B 0,C 180,E1 -17557.273,E2 -17557.273} C_VEL
LIN {X 0,Y 277.505,Z 549.916,A -85,B 0,C 180,E1 -17560.213,E2 -17560.213} C_VEL
LIN {X 0,Y 277.434,Z 549.923,A -85,B 0,C 180,E1 -17564.676,E2 -17564.676} C_VEL
LIN {X 0,Y 277.345,Z 549.936,A -85,B 0,C 180,E1 -17569.236,E2 -17569.236} C_VEL
LIN {X 0,Y 277.319,Z 549.933,A -85,B 0,C 180,E1 -17574.172,E2 -17574.172} C_VEL
LIN {X 0,Y 277.324,Z 549.941,A -85,B 0,C 180,E1 -17577.506,E2 -17577.506} C_VEL
LIN {X 0,Y 277.273,Z 549.944,A -85,B 0,C 180,E1 -17580.483,E2 -17580.483} C_VEL
LIN {X 0,Y 277.249,Z 549.947,A -85,B 0,C 180,E1 -17583.898,E2 -17583.898} C_VEL
LIN {X 0,Y 277.267,Z 549.948,A -85,B 0,C 180,E1 -17587.472,E2 -17587.472} C_VEL
LIN {X 0,Y 277.213,Z 549.951,A -85,B 0,C 180,E1 -17591.238,E2 -17591.238} C_VEL
LIN {X 0,Y 277.22,Z 549.954,A -85,B 0,C 180,E1 -17595.225,E2 -17595.225} C_VEL
LIN {X 0,Y 277.227,Z 549.948,A -85,B 0,C 180,E1 -17599.514,E2 -17599.514} C_VEL
LIN {X 0,Y 277.272,Z 549.942,A -85,B 0,C 180,E1 -17602.532,E2 -17602.532} C_VEL
LIN {X 0,Y 277.252,Z 549.947,A -85,B 0,C 180,E1 -17606.106,E2 -17606.106} C_VEL
LIN {X 0,Y 277.267,Z 549.945,A -85,B 0,C 180,E1 -17609.54,E2 -17609.54} C_VEL
LIN {X 0,Y 277.365,Z 549.928,A -85,B 0,C 180,E1 -17612.866,E2 -17612.866} C_VEL
LIN {X 0,Y 277.303,Z 549.941,A -85,B 0,C 180,E1 -17616.078,E2 -17616.078} C_VEL
LIN {X 0,Y 277.331,Z 549.934,A -85,B 0,C 180,E1 -17620.766,E2 -17620.766} C_VEL
LIN {X 0,Y 277.413,Z 549.925,A -85,B 0,C 180,E1 -17625.224,E2 -17625.224} C_VEL
LIN {X 0,Y 276.79,Z 550.008,A -85,B 0,C 180,E1 -17626.436,E2 -17626.436} C_VEL
LIN {X 0,Y 273.999,Z 550.357,A -85,B 0,C 180,E1 -17628.412,E2 -17628.412} C_VEL
LIN {X 0,Y 271.624,Z 550.648,A -85,B 0,C 180,E1 -17630.018,E2 -17630.018} C_VEL
LIN {X 0,Y 270.624,Z 550.772,A -85,B 0,C 180,E1 -17631.261,E2 -17631.261} C_VEL
LIN {X 0,Y 270.554,Z 550.775,A -85,B 0,C 180,E1 -17631.682,E2 -17631.682} C_VEL
LIN {X 0,Y 270.545,Z 550.78,A -85,B 0,C 180,E1 -17634.036,E2 -17634.036} C_VEL
LIN {X 0,Y 270.794,Z 550.752,A -85,B 0,C 180,E1 -17638.514,E2 -17638.514} C_VEL
LIN {X 0,Y 270.794,Z 550.752,A -85,B 0,C 180,E1 -17641.488,E2 -17641.488} C_VEL
LIN {X 0,Y 270.62,Z 550.774,A -85,B 0,C 180,E1 -17647.462,E2 -17647.462} C_VEL
LIN {X 0,Y 270.451,Z 550.794,A -85,B 0,C 180,E1 -17650.481,E2 -17650.481} C_VEL
LIN {X 0,Y 270.412,Z 550.798,A -85,B 0,C 180,E1 -17655.065,E2 -17655.065} C_VEL
LIN {X 0,Y 270.309,Z 550.814,A -85,B 0,C 180,E1 -17659.756,E2 -17659.756} C_VEL
LIN {X 0,Y 270.247,Z 550.811,A -85,B 0,C 180,E1 -17664.589,E2 -17664.589} C_VEL
LIN {X 0,Y 270.279,Z 550.815,A -85,B 0,C 180,E1 -17667.909,E2 -17667.909} C_VEL
LIN {X 0,Y 270.193,Z 550.826,A -85,B 0,C 180,E1 -17671.348,E2 -17671.348} C_VEL
LIN {X 0,Y 270.211,Z 550.825,A -85,B 0,C 180,E1 -17674.905,E2 -17674.905} C_VEL
LIN {X 0,Y 270.206,Z 550.826,A -85,B 0,C 180,E1 -17678.71,E2 -17678.71} C_VEL
LIN {X 0,Y 270.18,Z 550.831,A -85,B 0,C 180,E1 -17682.558,E2 -17682.558} C_VEL
LIN {X 0,Y 270.173,Z 550.831,A -85,B 0,C 180,E1 -17686.75,E2 -17686.75} C_VEL
LIN {X 0,Y 270.231,Z 550.821,A -85,B 0,C 180,E1 -17691.282,E2 -17691.282} C_VEL
LIN {X 0,Y 270.299,Z 550.93,A -85,B 0,C 180,E1 -17695.415,E2 -17695.415} C_VEL
LIN {X 0,Y 272.622,Z 561.892,A -85,B 0,C 180,E1 -17699.391,E2 -17699.391} C_VEL
LIN {X 0,Y 274.124,Z 569.065,A -85,B 0,C 180,E1 -17701.845,E2 -17701.845} C_VEL
LIN {X 0,Y 277.546,Z 579.407,A -85,B 0,C 180,E1 -17702.469,E2 -17702.469} C_VEL
LIN {X 0,Y 282.578,Z 614.314,A -85,B 0,C 180,E1 -17703.95,E2 -17703.95} C_VEL
LIN {X 0,Y 280.531,Z 677.894,A -85,B 0,C 180,E1 -17705.729,E2 -17705.729} C_VEL
LIN {X 0,Y 279.561,Z 691.24,A -85,B 0,C 180,E1 -17706.379,E2 -17706.379} C_VEL
LIN {X 0,Y 278.326,Z 703.521,A -85,B 0,C 180,E1 -17707.251,E2 -17707.251} C_VEL
LIN {X 0,Y 276.892,Z 715.401,A -85,B 0,C 180,E1 -17708.404,E2 -17708.404} C_VEL
LIN {X 0,Y 275.217,Z 726.855,A -85,B 0,C 180,E1 -17709.832,E2 -17709.832} C_VEL
LIN {X 0,Y 273.695,Z 737.224,A -85,B 0,C 180,E1 -17711.47,E2 -17711.47} C_VEL
LIN {X 0,Y 272.421,Z 746.086,A -85,B 0,C 180,E1 -17713.214,E2 -17713.214} C_VEL
LIN {X 0,Y 270.976,Z 754.895,A -85,B 0,C 180,E1 -17715.35,E2 -17715.35} C_VEL
LIN {X 0,Y 269.748,Z 762.279,A -85,B 0,C 180,E1 -17717.586,E2 -17717.586} C_VEL
LIN {X 0,Y 269.109,Z 767.264,A -85,B 0,C 180,E1 -17719.464,E2 -17719.464} C_VEL
LIN {X 0,Y 268.551,Z 772.083,A -85,B 0,C 180,E1 -17721.722,E2 -17721.722} C_VEL
LIN {X 0,Y 268.301,Z 775.745,A -85,B 0,C 180,E1 -17723.984,E2 -17723.984} C_VEL
LIN {X 0,Y 268.181,Z 777.614,A -85,B 0,C 180,E1 -17725.489,E2 -17725.489} C_VEL
LIN {X 0,Y 268.189,Z 779.002,A -85,B 0,C 180,E1 -17726.994,E2 -17726.994} C_VEL
LIN {X 0,Y 268.193,Z 779.976,A -85,B 0,C 180,E1 -17728.496,E2 -17728.496} C_VEL
LIN {X 0,Y 268.202,Z 780.547,A -85,B 0,C 180,E1 -17729.998,E2 -17729.998} C_VEL
LIN {X 0,Y 268.183,Z 780.699,A -85,B 0,C 180,E1 -17731.5,E2 -17731.5} C_VEL
LIN {X 0,Y 268.16,Z 780.413,A -85,B 0,C 180,E1 -17733.002,E2 -17733.002} C_VEL
LIN {X 0,Y 268.226,Z 778.664,A -85,B 0,C 180,E1 -17736.014,E2 -17736.014} C_VEL
LIN {X 0,Y 268.427,Z 777.171,A -85,B 0,C 180,E1 -17737.52,E2 -17737.52} C_VEL
LIN {X 0,Y 268.977,Z 774.107,A -85,B 0,C 180,E1 -17739.776,E2 -17739.776} C_VEL
LIN {X 0,Y 269.837,Z 769.993,A -85,B 0,C 180,E1 -17742.024,E2 -17742.024} C_VEL
LIN {X 0,Y 271.029,Z 764.725,A -85,B 0,C 180,E1 -17744.259,E2 -17744.259} C_VEL
LIN {X 0,Y 272.754,Z 758.122,A -85,B 0,C 180,E1 -17746.463,E2 -17746.463} C_VEL
LIN {X 0,Y 274.37,Z 750.98,A -85,B 0,C 180,E1 -17748.412,E2 -17748.412} C_VEL
LIN {X 0,Y 276.549,Z 741.696,A -85,B 0,C 180,E1 -17750.45,E2 -17750.45} C_VEL
LIN {X 0,Y 278.782,Z 731.615,A -85,B 0,C 180,E1 -17752.216,E2 -17752.216} C_VEL
LIN {X 0,Y 281.023,Z 720.273,A -85,B 0,C 180,E1 -17753.78,E2 -17753.78} C_VEL
LIN {X 0,Y 283.039,Z 709.221,A -85,B 0,C 180,E1 -17754.966,E2 -17754.966} C_VEL
LIN {X 0,Y 284.783,Z 697.059,A -85,B 0,C 180,E1 -17755.977,E2 -17755.977} C_VEL
LIN {X 0,Y 286.313,Z 683.562,A -85,B 0,C 180,E1 -17756.759,E2 -17756.759} C_VEL
LIN {X 0,Y 287.282,Z 670.334,A -85,B 0,C 180,E1 -17757.251,E2 -17757.251} C_VEL
LIN {X 0,Y 289.551,Z 615.398,A -85,B 0,C 180,E1 -17758.783,E2 -17758.783} C_VEL
LIN {X 0,Y 287.252,Z 599.449,A -85,B 0,C 180,E1 -17759.649,E2 -17759.649} C_VEL
LIN {X 0,Y 285.66,Z 590.876,A -85,B 0,C 180,E1 -17760.177,E2 -17760.177} C_VEL
LIN {X 0,Y 280.457,Z 579.196,A -85,B 0,C 180,E1 -17761.389,E2 -17761.389} C_VEL
LIN {X 0,Y 276.155,Z 570.791,A -85,B 0,C 180,E1 -17762.412,E2 -17762.412} C_VEL
LIN {X 0,Y 274.377,Z 567.031,A -85,B 0,C 180,E1 -17762.914,E2 -17762.914} C_VEL
LIN {X 0,Y 272.294,Z 558.159,A -85,B 0,C 180,E1 -17766.857,E2 -17766.857} C_VEL
LIN {X 0,Y 270.225,Z 550.84,A -85,B 0,C 180,E1 -17770.516,E2 -17770.516} C_VEL
LIN {X 0,Y 270.169,Z 550.833,A -85,B 0,C 180,E1 -17774.613,E2 -17774.613} C_VEL
LIN {X 0,Y 270.218,Z 550.825,A -85,B 0,C 180,E1 -17778.956,E2 -17778.956} C_VEL
LIN {X 0,Y 270.233,Z 550.818,A -85,B 0,C 180,E1 -17783.261,E2 -17783.261} C_VEL
LIN {X 0,Y 270.197,Z 550.826,A -85,B 0,C 180,E1 -17786.891,E2 -17786.891} C_VEL
LIN {X 0,Y 270.221,Z 550.824,A -85,B 0,C 180,E1 -17790.385,E2 -17790.385} C_VEL
LIN {X 0,Y 270.255,Z 550.816,A -85,B 0,C 180,E1 -17793.762,E2 -17793.762} C_VEL
LIN {X 0,Y 270.223,Z 550.815,A -85,B 0,C 180,E1 -17797.037,E2 -17797.037} C_VEL
LIN {X 0,Y 270.292,Z 550.805,A -85,B 0,C 180,E1 -17800.243,E2 -17800.243} C_VEL
LIN {X 0,Y 270.393,Z 550.795,A -85,B 0,C 180,E1 -17804.934,E2 -17804.934} C_VEL
LIN {X 0,Y 270.432,Z 550.797,A -85,B 0,C 180,E1 -17809.518,E2 -17809.518} C_VEL
LIN {X 0,Y 270.6,Z 550.771,A -85,B 0,C 180,E1 -17812.538,E2 -17812.538} C_VEL
LIN {X 0,Y 270.78,Z 550.749,A -85,B 0,C 180,E1 -17818.512,E2 -17818.512} C_VEL
LIN {X 0,Y 270.78,Z 550.751,A -85,B 0,C 180,E1 -17821.486,E2 -17821.486} C_VEL
LIN {X 0,Y 270.601,Z 550.774,A -85,B 0,C 180,E1 -17827.461,E2 -17827.461} C_VEL
LIN {X 0,Y 270.431,Z 550.799,A -85,B 0,C 180,E1 -17830.481,E2 -17830.481} C_VEL
LIN {X 0,Y 270.388,Z 550.917,A -85,B 0,C 180,E1 -17833.815,E2 -17833.815} C_VEL
LIN {X 0,Y 271.848,Z 556.546,A -85,B 0,C 180,E1 -17836.763,E2 -17836.763} C_VEL
LIN {X 0,Y 274.146,Z 560.56,A -85,B 0,C 180,E1 -17837.338,E2 -17837.338} C_VEL
LIN {X 0,Y 281.048,Z 573.153,A -85,B 0,C 180,E1 -17838.97,E2 -17838.97} C_VEL
LIN {X 0,Y 287.226,Z 586.336,A -85,B 0,C 180,E1 -17840.378,E2 -17840.378} C_VEL
LIN {X 0,Y 290.415,Z 593.945,A -85,B 0,C 180,E1 -17841.093,E2 -17841.093} C_VEL
LIN {X 0,Y 287.267,Z 663.2,A -85,B 0,C 180,E1 -17843.043,E2 -17843.043} C_VEL
LIN {X 0,Y 286.181,Z 676.396,A -85,B 0,C 180,E1 -17843.682,E2 -17843.682} C_VEL
LIN {X 0,Y 284.771,Z 688.666,A -85,B 0,C 180,E1 -17844.544,E2 -17844.544} C_VEL
LIN {X 0,Y 283.025,Z 700.388,A -85,B 0,C 180,E1 -17845.657,E2 -17845.657} C_VEL
LIN {X 0,Y 281.167,Z 710.898,A -85,B 0,C 180,E1 -17846.939,E2 -17846.939} C_VEL
LIN {X 0,Y 279.013,Z 721.668,A -85,B 0,C 180,E1 -17848.592,E2 -17848.592} C_VEL
LIN {X 0,Y 276.895,Z 730.862,A -85,B 0,C 180,E1 -17850.353,E2 -17850.353} C_VEL
LIN {X 0,Y 274.725,Z 739.726,A -85,B 0,C 180,E1 -17852.494,E2 -17852.494} C_VEL
LIN {X 0,Y 272.979,Z 746.499,A -85,B 0,C 180,E1 -17854.532,E2 -17854.532} C_VEL
LIN {X 0,Y 271.23,Z 753.099,A -85,B 0,C 180,E1 -17857.043,E2 -17857.043} C_VEL
LIN {X 0,Y 269.924,Z 758.202,A -85,B 0,C 180,E1 -17859.652,E2 -17859.652} C_VEL
LIN {X 0,Y 269.134,Z 761.43,A -85,B 0,C 180,E1 -17861.9,E2 -17861.9} C_VEL
LIN {X 0,Y 268.344,Z 764.291,A -85,B 0,C 180,E1 -17865.001,E2 -17865.001} C_VEL
LIN {X 0,Y 267.974,Z 765.241,A -85,B 0,C 180,E1 -17867.25,E2 -17867.25} C_VEL
LIN {X 0,Y 267.832,Z 765.28,A -85,B 0,C 180,E1 -17869.548,E2 -17869.548} C_VEL
LIN {X 0,Y 267.86,Z 764.338,A -85,B 0,C 180,E1 -17871.916,E2 -17871.916} C_VEL
LIN {X 0,Y 268.189,Z 761.818,A -85,B 0,C 180,E1 -17874.797,E2 -17874.797} C_VEL
LIN {X 0,Y 268.744,Z 757.657,A -85,B 0,C 180,E1 -17877.681,E2 -17877.681} C_VEL
LIN {X 0,Y 269.491,Z 752.331,A -85,B 0,C 180,E1 -17880.3,E2 -17880.3} C_VEL
LIN {X 0,Y 270.462,Z 746.226,A -85,B 0,C 180,E1 -17882.585,E2 -17882.585} C_VEL
LIN {X 0,Y 271.675,Z 738.507,A -85,B 0,C 180,E1 -17884.878,E2 -17884.878} C_VEL
LIN {X 0,Y 273.081,Z 730.043,A -85,B 0,C 180,E1 -17886.894,E2 -17886.894} C_VEL
LIN {X 0,Y 274.609,Z 719.981,A -85,B 0,C 180,E1 -17888.81,E2 -17888.81} C_VEL
LIN {X 0,Y 276.233,Z 709.116,A -85,B 0,C 180,E1 -17890.458,E2 -17890.458} C_VEL
LIN {X 0,Y 277.584,Z 698.503,A -85,B 0,C 180,E1 -17891.743,E2 -17891.743} C_VEL
LIN {X 0,Y 278.906,Z 686.25,A -85,B 0,C 180,E1 -17892.887,E2 -17892.887} C_VEL
LIN {X 0,Y 279.975,Z 672.966,A -85,B 0,C 180,E1 -17893.797,E2 -17893.797} C_VEL
LIN {X 0,Y 280.755,Z 659.644,A -85,B 0,C 180,E1 -17894.392,E2 -17894.392} C_VEL
LIN {X 0,Y 283.06,Z 589.372,A -85,B 0,C 180,E1 -17896.325,E2 -17896.325} C_VEL
LIN {X 0,Y 281.5,Z 582.424,A -85,B 0,C 180,E1 -17896.663,E2 -17896.663} C_VEL
LIN {X 0,Y 273.349,Z 560.208,A -85,B 0,C 180,E1 -17898.062,E2 -17898.062} C_VEL
LIN {X 0,Y 271.145,Z 554.413,A -85,B 0,C 180,E1 -17898.48,E2 -17898.48} C_VEL
LIN {X 0,Y 270.469,Z 550.794,A -85,B 0,C 180,E1 -17899.938,E2 -17899.938} C_VEL
LIN {X 0,Y 270.599,Z 550.78,A -85,B 0,C 180,E1 -17902.541,E2 -17902.541} C_VEL
LIN {X 0,Y 270.784,Z 550.755,A -85,B 0,C 180,E1 -17908.515,E2 -17908.515} C_VEL
LIN {X 0,Y 270.785,Z 550.753,A -85,B 0,C 180,E1 -17911.489,E2 -17911.489} C_VEL
LIN {X 0,Y 270.606,Z 550.777,A -85,B 0,C 180,E1 -17917.463,E2 -17917.463} C_VEL
LIN {X 0,Y 270.44,Z 550.797,A -85,B 0,C 180,E1 -17920.483,E2 -17920.483} C_VEL
LIN {X 0,Y 270.402,Z 550.802,A -85,B 0,C 180,E1 -17925.067,E2 -17925.067} C_VEL
LIN {X 0,Y 270.302,Z 550.809,A -85,B 0,C 180,E1 -17929.758,E2 -17929.758} C_VEL
LIN {X 0,Y 270.274,Z 550.811,A -85,B 0,C 180,E1 -17934.588,E2 -17934.588} C_VEL
LIN {X 0,Y 270.271,Z 550.818,A -85,B 0,C 180,E1 -17937.911,E2 -17937.911} C_VEL
LIN {X 0,Y 270.186,Z 550.827,A -85,B 0,C 180,E1 -17941.35,E2 -17941.35} C_VEL
LIN {X 0,Y 270.203,Z 550.826,A -85,B 0,C 180,E1 -17944.907,E2 -17944.907} C_VEL
LIN {X 0,Y 270.2,Z 550.826,A -85,B 0,C 180,E1 -17948.712,E2 -17948.712} C_VEL
LIN {X 0,Y 270.175,Z 550.83,A -85,B 0,C 180,E1 -17953.252,E2 -17953.252} C_VEL
LIN {X 0,Y 270.178,Z 550.83,A -85,B 0,C 180,E1 -17957.444,E2 -17957.444} C_VEL
LIN {X 0,Y 270.211,Z 550.821,A -85,B 0,C 180,E1 -17961.376,E2 -17961.376} C_VEL
LIN {X 0,Y 270.207,Z 550.826,A -85,B 0,C 180,E1 -17965.096,E2 -17965.096} C_VEL
LIN {X 0,Y 270.206,Z 550.824,A -85,B 0,C 180,E1 -17969.132,E2 -17969.132} C_VEL
LIN {X 0,Y 270.271,Z 550.812,A -85,B 0,C 180,E1 -17972.147,E2 -17972.147} C_VEL
LIN {X 0,Y 270.244,Z 550.823,A -85,B 0,C 180,E1 -17975.539,E2 -17975.539} C_VEL
LIN {X 0,Y 270.268,Z 550.814,A -85,B 0,C 180,E1 -17980.243,E2 -17980.243} C_VEL
LIN {X 0,Y 270.384,Z 550.799,A -85,B 0,C 180,E1 -17984.935,E2 -17984.935} C_VEL
LIN {X 0,Y 270.42,Z 550.801,A -85,B 0,C 180,E1 -17989.519,E2 -17989.519} C_VEL
LIN {X 0,Y 270.554,Z 550.775,A -85,B 0,C 180,E1 -17991.682,E2 -17991.682} C_VEL
LIN {X 0,Y 269.9,Z 550.858,A -85,B 0,C 180,E1 -17992.923,E2 -17992.923} C_VEL
LIN {X 0,Y 267.027,Z 551.216,A -85,B 0,C 180,E1 -17994.945,E2 -17994.945} C_VEL
LIN {X 0,Y 264.653,Z 551.515,A -85,B 0,C 180,E1 -17996.59,E2 -17996.59} C_VEL
LIN {X 0,Y 263.742,Z 551.634,A -85,B 0,C 180,E1 -17997.865,E2 -17997.865} C_VEL
LIN {X 0,Y 263.727,Z 551.631,A -85,B 0,C 180,E1 -17998.295,E2 -17998.295} C_VEL
LIN {X 0,Y 263.759,Z 551.629,A -85,B 0,C 180,E1 -18001.528,E2 -18001.528} C_VEL
LIN {X 0,Y 263.582,Z 551.652,A -85,B 0,C 180,E1 -18007.662,E2 -18007.662} C_VEL
LIN {X 0,Y 263.383,Z 551.673,A -85,B 0,C 180,E1 -18010.766,E2 -18010.766} C_VEL
LIN {X 0,Y 263.36,Z 551.678,A -85,B 0,C 180,E1 -18015.478,E2 -18015.478} C_VEL
LIN {X 0,Y 263.271,Z 551.686,A -85,B 0,C 180,E1 -18020.307,E2 -18020.307} C_VEL
LIN {X 0,Y 263.202,Z 551.687,A -85,B 0,C 180,E1 -18025.293,E2 -18025.293} C_VEL
LIN {X 0,Y 263.175,Z 551.701,A -85,B 0,C 180,E1 -18028.731,E2 -18028.731} C_VEL
LIN {X 0,Y 263.142,Z 551.707,A -85,B 0,C 180,E1 -18032.288,E2 -18032.288} C_VEL
LIN {X 0,Y 263.173,Z 551.704,A -85,B 0,C 180,E1 -18035.981,E2 -18035.981} C_VEL
LIN {X 0,Y 263.114,Z 551.71,A -85,B 0,C 180,E1 -18039.872,E2 -18039.872} C_VEL
LIN {X 0,Y 263.131,Z 551.709,A -85,B 0,C 180,E1 -18043.983,E2 -18043.983} C_VEL
LIN {X 0,Y 263.133,Z 551.707,A -85,B 0,C 180,E1 -18048.406,E2 -18048.406} C_VEL
LIN {X 0,Y 263.174,Z 551.702,A -85,B 0,C 180,E1 -18052.103,E2 -18052.103} C_VEL
LIN {X 0,Y 263.235,Z 551.879,A -85,B 0,C 180,E1 -18054.962,E2 -18054.962} C_VEL
LIN {X 0,Y 265.785,Z 563.789,A -85,B 0,C 180,E1 -18059.399,E2 -18059.399} C_VEL
LIN {X 0,Y 266.883,Z 568.995,A -85,B 0,C 180,E1 -18061.181,E2 -18061.181} C_VEL
LIN {X 0,Y 271.161,Z 581.394,A -85,B 0,C 180,E1 -18061.973,E2 -18061.973} C_VEL
LIN {X 0,Y 275.965,Z 614.912,A -85,B 0,C 180,E1 -18063.437,E2 -18063.437} C_VEL
LIN {X 0,Y 273.827,Z 677.896,A -85,B 0,C 180,E1 -18065.247,E2 -18065.247} C_VEL
LIN {X 0,Y 272.754,Z 691.899,A -85,B 0,C 180,E1 -18065.954,E2 -18065.954} C_VEL
LIN {X 0,Y 271.507,Z 703.909,A -85,B 0,C 180,E1 -18066.848,E2 -18066.848} C_VEL
LIN {X 0,Y 270.045,Z 715.656,A -85,B 0,C 180,E1 -18068.028,E2 -18068.028} C_VEL
LIN {X 0,Y 268.32,Z 727.026,A -85,B 0,C 180,E1 -18069.491,E2 -18069.491} C_VEL
LIN {X 0,Y 266.754,Z 737.315,A -85,B 0,C 180,E1 -18071.169,E2 -18071.169} C_VEL
LIN {X 0,Y 265.363,Z 746.581,A -85,B 0,C 180,E1 -18073.06,E2 -18073.06} C_VEL
LIN {X 0,Y 263.83,Z 755.587,A -85,B 0,C 180,E1 -18075.339,E2 -18075.339} C_VEL
LIN {X 0,Y 262.595,Z 762.785,A -85,B 0,C 180,E1 -18077.635,E2 -18077.635} C_VEL
LIN {X 0,Y 261.857,Z 768.514,A -85,B 0,C 180,E1 -18079.951,E2 -18079.951} C_VEL
LIN {X 0,Y 261.362,Z 772.996,A -85,B 0,C 180,E1 -18082.271,E2 -18082.271} C_VEL
LIN {X 0,Y 261.135,Z 776.542,A -85,B 0,C 180,E1 -18084.749,E2 -18084.749} C_VEL
LIN {X 0,Y 261.103,Z 778.698,A -85,B 0,C 180,E1 -18086.912,E2 -18086.912} C_VEL
LIN {X 0,Y 261.121,Z 779.701,A -85,B 0,C 180,E1 -18088.456,E2 -18088.456} C_VEL
LIN {X 0,Y 261.128,Z 780.299,A -85,B 0,C 180,E1 -18089.998,E2 -18089.998} C_VEL
LIN {X 0,Y 261.11,Z 780.495,A -85,B 0,C 180,E1 -18091.54,E2 -18091.54} C_VEL
LIN {X 0,Y 261.056,Z 780.245,A -85,B 0,C 180,E1 -18093.084,E2 -18093.084} C_VEL
LIN {X 0,Y 261.087,Z 779.312,A -85,B 0,C 180,E1 -18095.135,E2 -18095.135} C_VEL
LIN {X 0,Y 261.363,Z 777.098,A -85,B 0,C 180,E1 -18097.724,E2 -18097.724} C_VEL
LIN {X 0,Y 261.973,Z 774.078,A -85,B 0,C 180,E1 -18100.04,E2 -18100.04} C_VEL
LIN {X 0,Y 262.859,Z 770.031,A -85,B 0,C 180,E1 -18102.348,E2 -18102.348} C_VEL
LIN {X 0,Y 264.158,Z 764.854,A -85,B 0,C 180,E1 -18104.638,E2 -18104.638} C_VEL
LIN {X 0,Y 265.955,Z 758.36,A -85,B 0,C 180,E1 -18106.896,E2 -18106.896} C_VEL
LIN {X 0,Y 268.013,Z 749.818,A -85,B 0,C 180,E1 -18109.261,E2 -18109.261} C_VEL
LIN {X 0,Y 270.367,Z 740.324,A -85,B 0,C 180,E1 -18111.339,E2 -18111.339} C_VEL
LIN {X 0,Y 272.823,Z 729.89,A -85,B 0,C 180,E1 -18113.129,E2 -18113.129} C_VEL
LIN {X 0,Y 275.193,Z 718.237,A -85,B 0,C 180,E1 -18114.718,E2 -18114.718} C_VEL
LIN {X 0,Y 277.284,Z 706.735,A -85,B 0,C 180,E1 -18115.924,E2 -18115.924} C_VEL
LIN {X 0,Y 279.009,Z 694.999,A -85,B 0,C 180,E1 -18116.859,E2 -18116.859} C_VEL
LIN {X 0,Y 280.474,Z 681.772,A -85,B 0,C 180,E1 -18117.615,E2 -18117.615} C_VEL
LIN {X 0,Y 281.39,Z 668.999,A -85,B 0,C 180,E1 -18118.073,E2 -18118.073} C_VEL
LIN {X 0,Y 283.641,Z 616.142,A -85,B 0,C 180,E1 -18119.584,E2 -18119.584} C_VEL
LIN {X 0,Y 281.578,Z 601.42,A -85,B 0,C 180,E1 -18120.409,E2 -18120.409} C_VEL
LIN {X 0,Y 280.22,Z 593.985,A -85,B 0,C 180,E1 -18120.884,E2 -18120.884} C_VEL
LIN {X 0,Y 275.408,Z 582.917,A -85,B 0,C 180,E1 -18122.078,E2 -18122.078} C_VEL
LIN {X 0,Y 271.338,Z 574.943,A -85,B 0,C 180,E1 -18123.085,E2 -18123.085} C_VEL
LIN {X 0,Y 267.142,Z 566.746,A -85,B 0,C 180,E1 -18124.245,E2 -18124.245} C_VEL
LIN {X 0,Y 265.458,Z 559.797,A -85,B 0,C 180,E1 -18127.509,E2 -18127.509} C_VEL
LIN {X 0,Y 263.755,Z 553.78,A -85,B 0,C 180,E1 -18130.637,E2 -18130.637} C_VEL
LIN {X 0,Y 263.144,Z 551.713,A -85,B 0,C 180,E1 -18131.886,E2 -18131.886} C_VEL
LIN {X 0,Y 263.13,Z 551.713,A -85,B 0,C 180,E1 -18136.146,E2 -18136.146} C_VEL
LIN {X 0,Y 263.133,Z 551.704,A -85,B 0,C 180,E1 -18140.132,E2 -18140.132} C_VEL
LIN {X 0,Y 263.182,Z 551.703,A -85,B 0,C 180,E1 -18144.02,E2 -18144.02} C_VEL
LIN {X 0,Y 263.126,Z 551.709,A -85,B 0,C 180,E1 -18147.71,E2 -18147.71} C_VEL
LIN {X 0,Y 263.193,Z 551.697,A -85,B 0,C 180,E1 -18151.781,E2 -18151.781} C_VEL
LIN {X 0,Y 263.217,Z 551.696,A -85,B 0,C 180,E1 -18155.199,E2 -18155.199} C_VEL
LIN {X 0,Y 263.254,Z 551.684,A -85,B 0,C 180,E1 -18159.692,E2 -18159.692} C_VEL
LIN {X 0,Y 263.341,Z 551.672,A -85,B 0,C 180,E1 -18164.521,E2 -18164.521} C_VEL
LIN {X 0,Y 263.364,Z 551.675,A -85,B 0,C 180,E1 -18169.233,E2 -18169.233} C_VEL
LIN {X 0,Y 263.562,Z 551.647,A -85,B 0,C 180,E1 -18172.337,E2 -18172.337} C_VEL
LIN {X 0,Y 263.744,Z 551.625,A -85,B 0,C 180,E1 -18178.472,E2 -18178.472} C_VEL
LIN {X 0,Y 263.746,Z 551.627,A -85,B 0,C 180,E1 -18181.526,E2 -18181.526} C_VEL
LIN {X 0,Y 263.562,Z 551.651,A -85,B 0,C 180,E1 -18187.661,E2 -18187.661} C_VEL
LIN {X 0,Y 263.363,Z 551.681,A -85,B 0,C 180,E1 -18190.765,E2 -18190.765} C_VEL
LIN {X 0,Y 263.316,Z 551.726,A -85,B 0,C 180,E1 -18192.524,E2 -18192.524} C_VEL
LIN {X 0,Y 264.68,Z 556.823,A -85,B 0,C 180,E1 -18195.398,E2 -18195.398} C_VEL
LIN {X 0,Y 267.068,Z 560.936,A -85,B 0,C 180,E1 -18196.039,E2 -18196.039} C_VEL
LIN {X 0,Y 272.549,Z 570.352,A -85,B 0,C 180,E1 -18197.437,E2 -18197.437} C_VEL
LIN {X 0,Y 279.192,Z 583.508,A -85,B 0,C 180,E1 -18199.053,E2 -18199.053} C_VEL
LIN {X 0,Y 284.573,Z 596.21,A -85,B 0,C 180,E1 -18200.336,E2 -18200.336} C_VEL
LIN {X 0,Y 281.369,Z 663.235,A -85,B 0,C 180,E1 -18202.256,E2 -18202.256} C_VEL
LIN {X 0,Y 280.203,Z 676.328,A -85,B 0,C 180,E1 -18202.892,E2 -18202.892} C_VEL
LIN {X 0,Y 278.722,Z 688.875,A -85,B 0,C 180,E1 -18203.793,E2 -18203.793} C_VEL
LIN {X 0,Y 276.835,Z 700.777,A -85,B 0,C 180,E1 -18204.946,E2 -18204.946} C_VEL
LIN {X 0,Y 274.666,Z 712.444,A -85,B 0,C 180,E1 -18206.425,E2 -18206.425} C_VEL
LIN {X 0,Y 272.501,Z 722.581,A -85,B 0,C 180,E1 -18208.045,E2 -18208.045} C_VEL
LIN {X 0,Y 270.29,Z 731.557,A -85,B 0,C 180,E1 -18209.827,E2 -18209.827} C_VEL
LIN {X 0,Y 268.158,Z 739.798,A -85,B 0,C 180,E1 -18211.863,E2 -18211.863} C_VEL
LIN {X 0,Y 266.074,Z 747.485,A -85,B 0,C 180,E1 -18214.249,E2 -18214.249} C_VEL
LIN {X 0,Y 264.545,Z 752.865,A -85,B 0,C 180,E1 -18216.364,E2 -18216.364} C_VEL
LIN {X 0,Y 263.355,Z 757.165,A -85,B 0,C 180,E1 -18218.501,E2 -18218.501} C_VEL
LIN {X 0,Y 262.712,Z 759.533,A -85,B 0,C 180,E1 -18219.943,E2 -18219.943} C_VEL
LIN {X 0,Y 261.965,Z 762.291,A -85,B 0,C 180,E1 -18222.12,E2 -18222.12} C_VEL
LIN {X 0,Y 261.37,Z 764.235,A -85,B 0,C 180,E1 -18224.355,E2 -18224.355} C_VEL
LIN {X 0,Y 260.965,Z 765.335,A -85,B 0,C 180,E1 -18226.645,E2 -18226.645} C_VEL
LIN {X 0,Y 260.728,Z 765.449,A -85,B 0,C 180,E1 -18229.693,E2 -18229.693} C_VEL
LIN {X 0,Y 260.772,Z 764.624,A -85,B 0,C 180,E1 -18231.697,E2 -18231.697} C_VEL
LIN {X 0,Y 260.938,Z 762.943,A -85,B 0,C 180,E1 -18233.9,E2 -18233.9} C_VEL
LIN {X 0,Y 261.39,Z 759.889,A -85,B 0,C 180,E1 -18236.458,E2 -18236.458} C_VEL
LIN {X 0,Y 262.085,Z 754.857,A -85,B 0,C 180,E1 -18239.372,E2 -18239.372} C_VEL
LIN {X 0,Y 263.014,Z 749.015,A -85,B 0,C 180,E1 -18241.857,E2 -18241.857} C_VEL
LIN {X 0,Y 264.243,Z 741.56,A -85,B 0,C 180,E1 -18244.336,E2 -18244.336} C_VEL
LIN {X 0,Y 265.715,Z 732.786,A -85,B 0,C 180,E1 -18246.628,E2 -18246.628} C_VEL
LIN {X 0,Y 267.255,Z 723.314,A -85,B 0,C 180,E1 -18248.603,E2 -18248.603} C_VEL
LIN {X 0,Y 268.937,Z 712.806,A -85,B 0,C 180,E1 -18250.359,E2 -18250.359} C_VEL
LIN {X 0,Y 270.445,Z 701.643,A -85,B 0,C 180,E1 -18251.832,E2 -18251.832} C_VEL
LIN {X 0,Y 271.844,Z 689.843,A -85,B 0,C 180,E1 -18253.048,E2 -18253.048} C_VEL
LIN {X 0,Y 273.011,Z 677.095,A -85,B 0,C 180,E1 -18254.033,E2 -18254.033} C_VEL
LIN {X 0,Y 273.908,Z 664.261,A -85,B 0,C 180,E1 -18254.707,E2 -18254.707} C_VEL
LIN {X 0,Y 274.706,Z 642.652,A -85,B 0,C 180,E1 -18255.377,E2 -18255.377} C_VEL
LIN {X 0,Y 276.376,Z 589.841,A -85,B 0,C 180,E1 -18256.866,E2 -18256.866} C_VEL
LIN {X 0,Y 275.026,Z 584.359,A -85,B 0,C 180,E1 -18257.152,E2 -18257.152} C_VEL
LIN {X 0,Y 267.197,Z 563.012,A -85,B 0,C 180,E1 -18258.543,E2 -18258.543} C_VEL
LIN {X 0,Y 263.95,Z 554.587,A -85,B 0,C 180,E1 -18259.173,E2 -18259.173} C_VEL
LIN {X 0,Y 263.466,Z 551.668,A -85,B 0,C 180,E1 -18260.444,E2 -18260.444} C_VEL
LIN {X 0,Y 263.508,Z 551.663,A -85,B 0,C 180,E1 -18263.878,E2 -18263.878} C_VEL
LIN {X 0,Y 263.749,Z 551.631,A -85,B 0,C 180,E1 -18268.475,E2 -18268.475} C_VEL
LIN {X 0,Y 263.749,Z 551.629,A -85,B 0,C 180,E1 -18271.529,E2 -18271.529} C_VEL
LIN {X 0,Y 263.568,Z 551.653,A -85,B 0,C 180,E1 -18277.664,E2 -18277.664} C_VEL
LIN {X 0,Y 263.373,Z 551.679,A -85,B 0,C 180,E1 -18280.768,E2 -18280.768} C_VEL
LIN {X 0,Y 263.35,Z 551.68,A -85,B 0,C 180,E1 -18285.48,E2 -18285.48} C_VEL
LIN {X 0,Y 263.264,Z 551.685,A -85,B 0,C 180,E1 -18290.309,E2 -18290.309} C_VEL
LIN {X 0,Y 263.208,Z 551.696,A -85,B 0,C 180,E1 -18295.293,E2 -18295.293} C_VEL
LIN {X 0,Y 263.167,Z 551.704,A -85,B 0,C 180,E1 -18298.733,E2 -18298.733} C_VEL
LIN {X 0,Y 263.134,Z 551.701,A -85,B 0,C 180,E1 -18302.29,E2 -18302.29} C_VEL
LIN {X 0,Y 263.184,Z 551.701,A -85,B 0,C 180,E1 -18306.765,E2 -18306.765} C_VEL
LIN {X 0,Y 263.128,Z 551.706,A -85,B 0,C 180,E1 -18311.596,E2 -18311.596} C_VEL
LIN {X 0,Y 263.132,Z 551.706,A -85,B 0,C 180,E1 -18316.019,E2 -18316.019} C_VEL
LIN {X 0,Y 263.11,Z 551.701,A -85,B 0,C 180,E1 -18320.129,E2 -18320.129} C_VEL
LIN {X 0,Y 263.168,Z 551.702,A -85,B 0,C 180,E1 -18324.02,E2 -18324.02} C_VEL
LIN {X 0,Y 263.138,Z 551.706,A -85,B 0,C 180,E1 -18327.714,E2 -18327.714} C_VEL
LIN {X 0,Y 263.207,Z 551.693,A -85,B 0,C 180,E1 -18331.785,E2 -18331.785} C_VEL
LIN {X 0,Y 263.207,Z 551.696,A -85,B 0,C 180,E1 -18335.214,E2 -18335.214} C_VEL
LIN {X 0,Y 263.245,Z 551.692,A -85,B 0,C 180,E1 -18339.693,E2 -18339.693} C_VEL
LIN {X 0,Y 263.331,Z 551.677,A -85,B 0,C 180,E1 -18344.522,E2 -18344.522} C_VEL
LIN {X 0,Y 263.362,Z 551.678,A -85,B 0,C 180,E1 -18349.235,E2 -18349.235} C_VEL
LIN {X 0,Y 263.566,Z 551.646,A -85,B 0,C 180,E1 -18352.339,E2 -18352.339} C_VEL
LIN {X 0,Y 263.727,Z 551.631,A -85,B 0,C 180,E1 -18358.295,E2 -18358.295} C_VEL
LIN {X 0,Y 263.161,Z 551.707,A -85,B 0,C 180,E1 -18359.569,E2 -18359.569} C_VEL
LIN {X 0,Y 261.517,Z 551.913,A -85,B 0,C 180,E1 -18360.817,E2 -18360.817} C_VEL
LIN {X 0,Y 257.523,Z 552.403,A -85,B 0,C 180,E1 -18363.324,E2 -18363.324} C_VEL
LIN {X 0,Y 256.428,Z 552.536,A -85,B 0,C 180,E1 -18364.637,E2 -18364.637} C_VEL
LIN {X 0,Y 256.363,Z 552.543,A -85,B 0,C 180,E1 -18365.083,E2 -18365.083} C_VEL
LIN {X 0,Y 256.549,Z 552.53,A -85,B 0,C 180,E1 -18367.873,E2 -18367.873} C_VEL
LIN {X 0,Y 256.319,Z 552.553,A -85,B 0,C 180,E1 -18371.066,E2 -18371.066} C_VEL
LIN {X 0,Y 256.309,Z 552.559,A -85,B 0,C 180,E1 -18375.915,E2 -18375.915} C_VEL
LIN {X 0,Y 256.171,Z 552.568,A -85,B 0,C 180,E1 -18380.896,E2 -18380.896} C_VEL
LIN {X 0,Y 256.18,Z 552.56,A -85,B 0,C 180,E1 -18385.13,E2 -18385.13} C_VEL
LIN {X 0,Y 256.113,Z 552.581,A -85,B 0,C 180,E1 -18389.601,E2 -18389.601} C_VEL
LIN {X 0,Y 256.085,Z 552.584,A -85,B 0,C 180,E1 -18393.291,E2 -18393.291} C_VEL
LIN {X 0,Y 256.125,Z 552.58,A -85,B 0,C 180,E1 -18397.271,E2 -18397.271} C_VEL
LIN {X 0,Y 256.063,Z 552.587,A -85,B 0,C 180,E1 -18401.203,E2 -18401.203} C_VEL
LIN {X 0,Y 256.053,Z 552.585,A -85,B 0,C 180,E1 -18405.532,E2 -18405.532} C_VEL
LIN {X 0,Y 256.065,Z 552.586,A -85,B 0,C 180,E1 -18408.796,E2 -18408.796} C_VEL
LIN {X 0,Y 256.153,Z 552.579,A -85,B 0,C 180,E1 -18412.869,E2 -18412.869} C_VEL
LIN {X 0,Y 256.195,Z 552.754,A -85,B 0,C 180,E1 -18414.461,E2 -18414.461} C_VEL
LIN {X 0,Y 258.307,Z 562.651,A -85,B 0,C 180,E1 -18418.282,E2 -18418.282} C_VEL
LIN {X 0,Y 259.508,Z 568.467,A -85,B 0,C 180,E1 -18420.435,E2 -18420.435} C_VEL
LIN {X 0,Y 264.798,Z 583.51,A -85,B 0,C 180,E1 -18421.46,E2 -18421.46} C_VEL
LIN {X 0,Y 269.348,Z 615.625,A -85,B 0,C 180,E1 -18422.906,E2 -18422.906} C_VEL
LIN {X 0,Y 267.158,Z 677.841,A -85,B 0,C 180,E1 -18424.742,E2 -18424.742} C_VEL
LIN {X 0,Y 266.13,Z 691.047,A -85,B 0,C 180,E1 -18425.42,E2 -18425.42} C_VEL
LIN {X 0,Y 264.844,Z 703.26,A -85,B 0,C 180,E1 -18426.334,E2 -18426.334} C_VEL
LIN {X 0,Y 263.207,Z 715.896,A -85,B 0,C 180,E1 -18427.633,E2 -18427.633} C_VEL
LIN {X 0,Y 261.432,Z 727.187,A -85,B 0,C 180,E1 -18429.131,E2 -18429.131} C_VEL
LIN {X 0,Y 259.822,Z 737.391,A -85,B 0,C 180,E1 -18430.852,E2 -18430.852} C_VEL
LIN {X 0,Y 258.258,Z 747.443,A -85,B 0,C 180,E1 -18432.988,E2 -18432.988} C_VEL
LIN {X 0,Y 256.933,Z 754.894,A -85,B 0,C 180,E1 -18434.936,E2 -18434.936} C_VEL
LIN {X 0,Y 255.623,Z 762.206,A -85,B 0,C 180,E1 -18437.292,E2 -18437.292} C_VEL
LIN {X 0,Y 254.825,Z 768.021,A -85,B 0,C 180,E1 -18439.671,E2 -18439.671} C_VEL
LIN {X 0,Y 254.317,Z 772.572,A -85,B 0,C 180,E1 -18442.056,E2 -18442.056} C_VEL
LIN {X 0,Y 254.026,Z 776.493,A -85,B 0,C 180,E1 -18444.877,E2 -18444.877} C_VEL
LIN {X 0,Y 254,Z 778.394,A -85,B 0,C 180,E1 -18446.825,E2 -18446.825} C_VEL
LIN {X 0,Y 254.05,Z 779.426,A -85,B 0,C 180,E1 -18448.413,E2 -18448.413} C_VEL
LIN {X 0,Y 254.056,Z 780.052,A -85,B 0,C 180,E1 -18449.998,E2 -18449.998} C_VEL
LIN {X 0,Y 254.016,Z 780.277,A -85,B 0,C 180,E1 -18451.583,E2 -18451.583} C_VEL
LIN {X 0,Y 253.956,Z 780.076,A -85,B 0,C 180,E1 -18453.171,E2 -18453.171} C_VEL
LIN {X 0,Y 253.992,Z 779.301,A -85,B 0,C 180,E1 -18455.036,E2 -18455.036} C_VEL
LIN {X 0,Y 254.32,Z 777.023,A -85,B 0,C 180,E1 -18457.94,E2 -18457.94} C_VEL
LIN {X 0,Y 254.946,Z 774.067,A -85,B 0,C 180,E1 -18460.32,E2 -18460.32} C_VEL
LIN {X 0,Y 255.889,Z 770.086,A -85,B 0,C 180,E1 -18462.69,E2 -18462.69} C_VEL
LIN {X 0,Y 257.302,Z 764.978,A -85,B 0,C 180,E1 -18465.037,E2 -18465.037} C_VEL
LIN {X 0,Y 259.156,Z 758.589,A -85,B 0,C 180,E1 -18467.353,E2 -18467.353} C_VEL
LIN {X 0,Y 261.185,Z 750.657,A -85,B 0,C 180,E1 -18469.644,E2 -18469.644} C_VEL
LIN {X 0,Y 263.323,Z 742.578,A -85,B 0,C 180,E1 -18471.527,E2 -18471.527} C_VEL
LIN {X 0,Y 265.774,Z 732.811,A -85,B 0,C 180,E1 -18473.367,E2 -18473.367} C_VEL
LIN {X 0,Y 268.189,Z 722.001,A -85,B 0,C 180,E1 -18474.994,E2 -18474.994} C_VEL
LIN {X 0,Y 270.683,Z 709.76,A -85,B 0,C 180,E1 -18476.397,E2 -18476.397} C_VEL
LIN {X 0,Y 272.557,Z 697.954,A -85,B 0,C 180,E1 -18477.443,E2 -18477.443} C_VEL
LIN {X 0,Y 274.197,Z 685.255,A -85,B 0,C 180,E1 -18478.251,E2 -18478.251} C_VEL
LIN {X 0,Y 275.397,Z 671.976,A -85,B 0,C 180,E1 -18478.793,E2 -18478.793} C_VEL
LIN {X 0,Y 277.896,Z 617.604,A -85,B 0,C 180,E1 -18480.382,E2 -18480.382} C_VEL
LIN {X 0,Y 275.931,Z 603.023,A -85,B 0,C 180,E1 -18481.233,E2 -18481.233} C_VEL
LIN {X 0,Y 274.855,Z 597.006,A -85,B 0,C 180,E1 -18481.637,E2 -18481.637} C_VEL
LIN {X 0,Y 270.348,Z 586.542,A -85,B 0,C 180,E1 -18482.807,E2 -18482.807} C_VEL
LIN {X 0,Y 264.911,Z 575.818,A -85,B 0,C 180,E1 -18484.252,E2 -18484.252} C_VEL
LIN {X 0,Y 261.911,Z 570.471,A -85,B 0,C 180,E1 -18485.072,E2 -18485.072} C_VEL
LIN {X 0,Y 259.95,Z 566.543,A -85,B 0,C 180,E1 -18485.67,E2 -18485.67} C_VEL
LIN {X 0,Y 258.194,Z 559.676,A -85,B 0,C 180,E1 -18489.145,E2 -18489.145} C_VEL
LIN {X 0,Y 256.074,Z 552.594,A -85,B 0,C 180,E1 -18493.241,E2 -18493.241} C_VEL
LIN {X 0,Y 256.086,Z 552.585,A -85,B 0,C 180,E1 -18497.812,E2 -18497.812} C_VEL
LIN {X 0,Y 256.094,Z 552.585,A -85,B 0,C 180,E1 -18500.861,E2 -18500.861} C_VEL
LIN {X 0,Y 256.114,Z 552.58,A -85,B 0,C 180,E1 -18504.811,E2 -18504.811} C_VEL
LIN {X 0,Y 256.085,Z 552.58,A -85,B 0,C 180,E1 -18508.57,E2 -18508.57} C_VEL
LIN {X 0,Y 256.134,Z 552.572,A -85,B 0,C 180,E1 -18512.194,E2 -18512.194} C_VEL
LIN {X 0,Y 256.158,Z 552.57,A -85,B 0,C 180,E1 -18515.697,E2 -18515.697} C_VEL
LIN {X 0,Y 256.158,Z 552.574,A -85,B 0,C 180,E1 -18519.103,E2 -18519.103} C_VEL
LIN {X 0,Y 256.29,Z 552.55,A -85,B 0,C 180,E1 -18524.084,E2 -18524.084} C_VEL
LIN {X 0,Y 256.3,Z 552.552,A -85,B 0,C 180,E1 -18528.933,E2 -18528.933} C_VEL
LIN {X 0,Y 256.529,Z 552.522,A -85,B 0,C 180,E1 -18532.126,E2 -18532.126} C_VEL
LIN {X 0,Y 256.707,Z 552.502,A -85,B 0,C 180,E1 -18538.43,E2 -18538.43} C_VEL
LIN {X 0,Y 256.71,Z 552.503,A -85,B 0,C 180,E1 -18541.568,E2 -18541.568} C_VEL
LIN {X 0,Y 256.529,Z 552.528,A -85,B 0,C 180,E1 -18547.872,E2 -18547.872} C_VEL
LIN {X 0,Y 256.322,Z 552.621,A -85,B 0,C 180,E1 -18551.165,E2 -18551.165} C_VEL
LIN {X 0,Y 257.578,Z 557.303,A -85,B 0,C 180,E1 -18553.912,E2 -18553.912} C_VEL
LIN {X 0,Y 259.985,Z 561.248,A -85,B 0,C 180,E1 -18554.614,E2 -18554.614} C_VEL
LIN {X 0,Y 266.134,Z 571.511,A -85,B 0,C 180,E1 -18556.294,E2 -18556.294} C_VEL
LIN {X 0,Y 272.676,Z 584.05,A -85,B 0,C 180,E1 -18557.989,E2 -18557.989} C_VEL
LIN {X 0,Y 278.719,Z 597.972,A -85,B 0,C 180,E1 -18559.513,E2 -18559.513} C_VEL
LIN {X 0,Y 275.423,Z 664.195,A -85,B 0,C 180,E1 -18561.469,E2 -18561.469} C_VEL
LIN {X 0,Y 274.227,Z 676.966,A -85,B 0,C 180,E1 -18562.111,E2 -18562.111} C_VEL
LIN {X 0,Y 272.645,Z 689.635,A -85,B 0,C 180,E1 -18563.046,E2 -18563.046} C_VEL
LIN {X 0,Y 270.816,Z 700.586,A -85,B 0,C 180,E1 -18564.124,E2 -18564.124} C_VEL
LIN {X 0,Y 268.606,Z 711.967,A -85,B 0,C 180,E1 -18565.576,E2 -18565.576} C_VEL
LIN {X 0,Y 266.221,Z 722.639,A -85,B 0,C 180,E1 -18567.3,E2 -18567.3} C_VEL
LIN {X 0,Y 263.672,Z 732.501,A -85,B 0,C 180,E1 -18569.324,E2 -18569.324} C_VEL
LIN {X 0,Y 261.643,Z 739.908,A -85,B 0,C 180,E1 -18571.211,E2 -18571.211} C_VEL
LIN {X 0,Y 259.639,Z 746.861,A -85,B 0,C 180,E1 -18573.391,E2 -18573.391} C_VEL
LIN {X 0,Y 257.644,Z 753.53,A -85,B 0,C 180,E1 -18576.049,E2 -18576.049} C_VEL
LIN {X 0,Y 256.393,Z 757.76,A -85,B 0,C 180,E1 -18578.251,E2 -18578.251} C_VEL
LIN {X 0,Y 255.362,Z 761.195,A -85,B 0,C 180,E1 -18580.598,E2 -18580.598} C_VEL
LIN {X 0,Y 254.932,Z 762.673,A -85,B 0,C 180,E1 -18581.902,E2 -18581.902} C_VEL
LIN {X 0,Y 254.342,Z 764.467,A -85,B 0,C 180,E1 -18584.078,E2 -18584.078} C_VEL
LIN {X 0,Y 253.941,Z 765.495,A -85,B 0,C 180,E1 -18586.224,E2 -18586.224} C_VEL
LIN {X 0,Y 253.709,Z 765.806,A -85,B 0,C 180,E1 -18588.41,E2 -18588.41} C_VEL
LIN {X 0,Y 253.629,Z 765.218,A -85,B 0,C 180,E1 -18590.883,E2 -18590.883} C_VEL
LIN {X 0,Y 253.777,Z 763.573,A -85,B 0,C 180,E1 -18593.427,E2 -18593.427} C_VEL
LIN {X 0,Y 254.303,Z 760.168,A -85,B 0,C 180,E1 -18596.449,E2 -18596.449} C_VEL
LIN {X 0,Y 254.822,Z 756.456,A -85,B 0,C 180,E1 -18598.756,E2 -18598.756} C_VEL
LIN {X 0,Y 255.764,Z 750.48,A -85,B 0,C 180,E1 -18601.558,E2 -18601.558} C_VEL
LIN {X 0,Y 256.957,Z 743.498,A -85,B 0,C 180,E1 -18604.051,E2 -18604.051} C_VEL
LIN {X 0,Y 258.31,Z 735.693,A -85,B 0,C 180,E1 -18606.272,E2 -18606.272} C_VEL
LIN {X 0,Y 259.912,Z 726.478,A -85,B 0,C 180,E1 -18608.384,E2 -18608.384} C_VEL
LIN {X 0,Y 261.622,Z 716.132,A -85,B 0,C 180,E1 -18610.268,E2 -18610.268} C_VEL
LIN {X 0,Y 263.274,Z 704.697,A -85,B 0,C 180,E1 -18611.924,E2 -18611.924} C_VEL
LIN {X 0,Y 264.836,Z 692.372,A -85,B 0,C 180,E1 -18613.302,E2 -18613.302} C_VEL
LIN {X 0,Y 266.16,Z 679.161,A -85,B 0,C 180,E1 -18614.397,E2 -18614.397} C_VEL
LIN {X 0,Y 267.146,Z 666.319,A -85,B 0,C 180,E1 -18615.138,E2 -18615.138} C_VEL
LIN {X 0,Y 267.806,Z 650.722,A -85,B 0,C 180,E1 -18615.678,E2 -18615.678} C_VEL
LIN {X 0,Y 269.816,Z 590.93,A -85,B 0,C 180,E1 -18617.401,E2 -18617.401} C_VEL
LIN {X 0,Y 268.458,Z 585.962,A -85,B 0,C 180,E1 -18617.682,E2 -18617.682} C_VEL
LIN {X 0,Y 261.154,Z 566.003,A -85,B 0,C 180,E1 -18619.019,E2 -18619.019} C_VEL
LIN {X 0,Y 256.837,Z 554.848,A -85,B 0,C 180,E1 -18619.857,E2 -18619.857} C_VEL
LIN {X 0,Y 256.468,Z 552.539,A -85,B 0,C 180,E1 -18620.863,E2 -18620.863} C_VEL
LIN {X 0,Y 256.48,Z 552.539,A -85,B 0,C 180,E1 -18623.71,E2 -18623.71} C_VEL
LIN {X 0,Y 256.712,Z 552.508,A -85,B 0,C 180,E1 -18628.433,E2 -18628.433} C_VEL
LIN {X 0,Y 256.712,Z 552.506,A -85,B 0,C 180,E1 -18631.571,E2 -18631.571} C_VEL
LIN {X 0,Y 256.536,Z 552.529,A -85,B 0,C 180,E1 -18637.875,E2 -18637.875} C_VEL
LIN {X 0,Y 256.309,Z 552.555,A -85,B 0,C 180,E1 -18641.068,E2 -18641.068} C_VEL
LIN {X 0,Y 256.3,Z 552.557,A -85,B 0,C 180,E1 -18645.917,E2 -18645.917} C_VEL
LIN {X 0,Y 256.167,Z 552.567,A -85,B 0,C 180,E1 -18650.897,E2 -18650.897} C_VEL
LIN {X 0,Y 256.189,Z 552.568,A -85,B 0,C 180,E1 -18655.14,E2 -18655.14} C_VEL
LIN {X 0,Y 256.105,Z 552.583,A -85,B 0,C 180,E1 -18659.603,E2 -18659.603} C_VEL
LIN {X 0,Y 256.069,Z 552.586,A -85,B 0,C 180,E1 -18663.295,E2 -18663.295} C_VEL
LIN {X 0,Y 256.117,Z 552.584,A -85,B 0,C 180,E1 -18667.273,E2 -18667.273} C_VEL
LIN {X 0,Y 256.058,Z 552.584,A -85,B 0,C 180,E1 -18671.205,E2 -18671.205} C_VEL
LIN {X 0,Y 256.066,Z 552.589,A -85,B 0,C 180,E1 -18675.531,E2 -18675.531} C_VEL
LIN {X 0,Y 256.059,Z 552.585,A -85,B 0,C 180,E1 -18678.799,E2 -18678.799} C_VEL
LIN {X 0,Y 256.135,Z 552.575,A -85,B 0,C 180,E1 -18682.869,E2 -18682.869} C_VEL
LIN {X 0,Y 256.073,Z 552.585,A -85,B 0,C 180,E1 -18686.709,E2 -18686.709} C_VEL
LIN {X 0,Y 256.12,Z 552.572,A -85,B 0,C 180,E1 -18690.402,E2 -18690.402} C_VEL
LIN {X 0,Y 256.177,Z 552.57,A -85,B 0,C 180,E1 -18694.872,E2 -18694.872} C_VEL
LIN {X 0,Y 256.155,Z 552.575,A -85,B 0,C 180,E1 -18699.105,E2 -18699.105} C_VEL
LIN {X 0,Y 256.266,Z 552.558,A -85,B 0,C 180,E1 -18704.084,E2 -18704.084} C_VEL
LIN {X 0,Y 256.297,Z 552.558,A -85,B 0,C 180,E1 -18707.329,E2 -18707.329} C_VEL
LIN {X 0,Y 256.523,Z 552.524,A -85,B 0,C 180,E1 -18712.127,E2 -18712.127} C_VEL
LIN {X 0,Y 256.505,Z 552.53,A -85,B 0,C 180,E1 -18716.86,E2 -18716.86} C_VEL
LIN {X 0,Y 256.773,Z 552.5,A -85,B 0,C 180,E1 -18720.001,E2 -18720.001} C_VEL
LIN {X 0,Y 256.506,Z 552.527,A -85,B 0,C 180,E1 -18723.142,E2 -18723.142} C_VEL
LIN {X 0,Y 256.363,Z 552.543,A -85,B 0,C 180,E1 -18725.083,E2 -18725.083} C_VEL
LIN {X 0,Y 255.752,Z 552.625,A -85,B 0,C 180,E1 -18726.397,E2 -18726.397} C_VEL
LIN {X 0,Y 252.886,Z 552.983,A -85,B 0,C 180,E1 -18728.538,E2 -18728.538} C_VEL
LIN {X 0,Y 250.402,Z 553.292,A -85,B 0,C 180,E1 -18730.28,E2 -18730.28} C_VEL
LIN {X 0,Y 249.319,Z 553.427,A -85,B 0,C 180,E1 -18731.633,E2 -18731.633} C_VEL
LIN {X 0,Y 249.224,Z 553.432,A -85,B 0,C 180,E1 -18732.092,E2 -18732.092} C_VEL
LIN {X 0,Y 249.228,Z 553.44,A -85,B 0,C 180,E1 -18736.503,E2 -18736.503} C_VEL
LIN {X 0,Y 249.093,Z 553.45,A -85,B 0,C 180,E1 -18741.518,E2 -18741.518} C_VEL
LIN {X 0,Y 249.126,Z 553.438,A -85,B 0,C 180,E1 -18745.475,E2 -18745.475} C_VEL
LIN {X 0,Y 249.083,Z 553.456,A -85,B 0,C 180,E1 -18748.989,E2 -18748.989} C_VEL
LIN {X 0,Y 249.042,Z 553.463,A -85,B 0,C 180,E1 -18752.425,E2 -18752.425} C_VEL
LIN {X 0,Y 249.067,Z 553.461,A -85,B 0,C 180,E1 -18756.34,E2 -18756.34} C_VEL
LIN {X 0,Y 249.015,Z 553.468,A -85,B 0,C 180,E1 -18760.477,E2 -18760.477} C_VEL
LIN {X 0,Y 249.004,Z 553.464,A -85,B 0,C 180,E1 -18764.88,E2 -18764.88} C_VEL
LIN {X 0,Y 249.018,Z 553.465,A -85,B 0,C 180,E1 -18767.361,E2 -18767.361} C_VEL
LIN {X 0,Y 249.047,Z 553.461,A -85,B 0,C 180,E1 -18771.621,E2 -18771.621} C_VEL
LIN {X 0,Y 249.155,Z 553.596,A -85,B 0,C 180,E1 -18773.935,E2 -18773.935} C_VEL
LIN {X 0,Y 251.253,Z 563.561,A -85,B 0,C 180,E1 -18777.893,E2 -18777.893} C_VEL
LIN {X 0,Y 252.286,Z 568.385,A -85,B 0,C 180,E1 -18779.722,E2 -18779.722} C_VEL
LIN {X 0,Y 258.525,Z 585.982,A -85,B 0,C 180,E1 -18780.948,E2 -18780.948} C_VEL
LIN {X 0,Y 262.736,Z 616.076,A -85,B 0,C 180,E1 -18782.338,E2 -18782.338} C_VEL
LIN {X 0,Y 260.546,Z 676.787,A -85,B 0,C 180,E1 -18784.167,E2 -18784.167} C_VEL
LIN {X 0,Y 259.515,Z 690.189,A -85,B 0,C 180,E1 -18784.857,E2 -18784.857} C_VEL
LIN {X 0,Y 258.142,Z 702.569,A -85,B 0,C 180,E1 -18785.788,E2 -18785.788} C_VEL
LIN {X 0,Y 256.573,Z 714.541,A -85,B 0,C 180,E1 -18787.023,E2 -18787.023} C_VEL
LIN {X 0,Y 254.818,Z 726.055,A -85,B 0,C 180,E1 -18788.563,E2 -18788.563} C_VEL
LIN {X 0,Y 253.095,Z 736.466,A -85,B 0,C 180,E1 -18790.322,E2 -18790.322} C_VEL
LIN {X 0,Y 251.68,Z 744.984,A -85,B 0,C 180,E1 -18792.109,E2 -18792.109} C_VEL
LIN {X 0,Y 250.03,Z 754.199,A -85,B 0,C 180,E1 -18794.51,E2 -18794.51} C_VEL
LIN {X 0,Y 248.662,Z 761.601,A -85,B 0,C 180,E1 -18796.93,E2 -18796.93} C_VEL
LIN {X 0,Y 247.811,Z 767.518,A -85,B 0,C 180,E1 -18799.375,E2 -18799.375} C_VEL
LIN {X 0,Y 247.267,Z 772.142,A -85,B 0,C 180,E1 -18801.828,E2 -18801.828} C_VEL
LIN {X 0,Y 246.948,Z 776.352,A -85,B 0,C 180,E1 -18804.934,E2 -18804.934} C_VEL
LIN {X 0,Y 246.901,Z 778.075,A -85,B 0,C 180,E1 -18806.734,E2 -18806.734} C_VEL
LIN {X 0,Y 246.957,Z 779.146,A -85,B 0,C 180,E1 -18808.367,E2 -18808.367} C_VEL
LIN {X 0,Y 246.985,Z 779.8,A -85,B 0,C 180,E1 -18809.998,E2 -18809.998} C_VEL
LIN {X 0,Y 246.923,Z 780.054,A -85,B 0,C 180,E1 -18811.629,E2 -18811.629} C_VEL
LIN {X 0,Y 246.859,Z 779.906,A -85,B 0,C 180,E1 -18813.262,E2 -18813.262} C_VEL
LIN {X 0,Y 246.884,Z 779.319,A -85,B 0,C 180,E1 -18814.897,E2 -18814.897} C_VEL
LIN {X 0,Y 247.274,Z 776.951,A -85,B 0,C 180,E1 -18818.168,E2 -18818.168} C_VEL
LIN {X 0,Y 247.926,Z 774.058,A -85,B 0,C 180,E1 -18820.615,E2 -18820.615} C_VEL
LIN {X 0,Y 248.931,Z 770.141,A -85,B 0,C 180,E1 -18823.051,E2 -18823.051} C_VEL
LIN {X 0,Y 250.453,Z 765.108,A -85,B 0,C 180,E1 -18825.458,E2 -18825.458} C_VEL
LIN {X 0,Y 252.378,Z 758.825,A -85,B 0,C 180,E1 -18827.835,E2 -18827.835} C_VEL
LIN {X 0,Y 254.425,Z 751.433,A -85,B 0,C 180,E1 -18830.083,E2 -18830.083} C_VEL
LIN {X 0,Y 256.751,Z 743.106,A -85,B 0,C 180,E1 -18832.107,E2 -18832.107} C_VEL
LIN {X 0,Y 259.62,Z 732.408,A -85,B 0,C 180,E1 -18834.167,E2 -18834.167} C_VEL
LIN {X 0,Y 262.134,Z 721.542,A -85,B 0,C 180,E1 -18835.826,E2 -18835.826} C_VEL
LIN {X 0,Y 264.735,Z 709.237,A -85,B 0,C 180,E1 -18837.252,E2 -18837.252} C_VEL
LIN {X 0,Y 266.72,Z 697.37,A -85,B 0,C 180,E1 -18838.311,E2 -18838.311} C_VEL
LIN {X 0,Y 268.413,Z 684.56,A -85,B 0,C 180,E1 -18839.131,E2 -18839.131} C_VEL
LIN {X 0,Y 269.613,Z 671.172,A -85,B 0,C 180,E1 -18839.685,E2 -18839.685} C_VEL
LIN {X 0,Y 272.163,Z 618.1,A -85,B 0,C 180,E1 -18841.28,E2 -18841.28} C_VEL
LIN {X 0,Y 270.151,Z 603.252,A -85,B 0,C 180,E1 -18842.189,E2 -18842.189} C_VEL
LIN {X 0,Y 269.353,Z 599.428,A -85,B 0,C 180,E1 -18842.477,E2 -18842.477} C_VEL
LIN {X 0,Y 264.699,Z 588.714,A -85,B 0,C 180,E1 -18843.761,E2 -18843.761} C_VEL
LIN {X 0,Y 258.069,Z 575.87,A -85,B 0,C 180,E1 -18845.639,E2 -18845.639} C_VEL
LIN {X 0,Y 255.054,Z 570.613,A -85,B 0,C 180,E1 -18846.539,E2 -18846.539} C_VEL
LIN {X 0,Y 252.666,Z 566.221,A -85,B 0,C 180,E1 -18847.317,E2 -18847.317} C_VEL
LIN {X 0,Y 250.914,Z 559.756,A -85,B 0,C 180,E1 -18850.863,E2 -18850.863} C_VEL
LIN {X 0,Y 249.007,Z 553.469,A -85,B 0,C 180,E1 -18854.874,E2 -18854.874} C_VEL
LIN {X 0,Y 249.026,Z 553.463,A -85,B 0,C 180,E1 -18857.364,E2 -18857.364} C_VEL
LIN {X 0,Y 249.041,Z 553.462,A -85,B 0,C 180,E1 -18861.621,E2 -18861.621} C_VEL
LIN {X 0,Y 249.054,Z 553.454,A -85,B 0,C 180,E1 -18865.64,E2 -18865.64} C_VEL
LIN {X 0,Y 249.044,Z 553.455,A -85,B 0,C 180,E1 -18869.471,E2 -18869.471} C_VEL
LIN {X 0,Y 249.065,Z 553.451,A -85,B 0,C 180,E1 -18873.16,E2 -18873.16} C_VEL
LIN {X 0,Y 249.07,Z 553.449,A -85,B 0,C 180,E1 -18876.731,E2 -18876.731} C_VEL
LIN {X 0,Y 249.101,Z 553.444,A -85,B 0,C 180,E1 -18880.21,E2 -18880.21} C_VEL
LIN {X 0,Y 249.232,Z 553.43,A -85,B 0,C 180,E1 -18883.62,E2 -18883.62} C_VEL
LIN {X 0,Y 249.243,Z 553.429,A -85,B 0,C 180,E1 -18888.615,E2 -18888.615} C_VEL
LIN {X 0,Y 249.474,Z 553.4,A -85,B 0,C 180,E1 -18891.902,E2 -18891.902} C_VEL
LIN {X 0,Y 249.431,Z 553.414,A -85,B 0,C 180,E1 -18896.769,E2 -18896.769} C_VEL
LIN {X 0,Y 249.726,Z 553.378,A -85,B 0,C 180,E1 -18899.999,E2 -18899.999} C_VEL
LIN {X 0,Y 249.452,Z 553.413,A -85,B 0,C 180,E1 -18903.229,E2 -18903.229} C_VEL
LIN {X 0,Y 249.471,Z 553.408,A -85,B 0,C 180,E1 -18908.097,E2 -18908.097} C_VEL
LIN {X 0,Y 249.405,Z 553.614,A -85,B 0,C 180,E1 -18909.733,E2 -18909.733} C_VEL
LIN {X 0,Y 250.399,Z 557.577,A -85,B 0,C 180,E1 -18912.237,E2 -18912.237} C_VEL
LIN {X 0,Y 252.934,Z 561.68,A -85,B 0,C 180,E1 -18913.047,E2 -18913.047} C_VEL
LIN {X 0,Y 257.219,Z 568.434,A -85,B 0,C 180,E1 -18914.336,E2 -18914.336} C_VEL
LIN {X 0,Y 263.372,Z 579.11,A -85,B 0,C 180,E1 -18916.072,E2 -18916.072} C_VEL
LIN {X 0,Y 269.706,Z 592.201,A -85,B 0,C 180,E1 -18917.792,E2 -18917.792} C_VEL
LIN {X 0,Y 273.036,Z 600.101,A -85,B 0,C 180,E1 -18918.665,E2 -18918.665} C_VEL
LIN {X 0,Y 269.696,Z 663.915,A -85,B 0,C 180,E1 -18920.587,E2 -18920.587} C_VEL
LIN {X 0,Y 268.416,Z 677.014,A -85,B 0,C 180,E1 -18921.252,E2 -18921.252} C_VEL
LIN {X 0,Y 266.752,Z 689.557,A -85,B 0,C 180,E1 -18922.187,E2 -18922.187} C_VEL
LIN {X 0,Y 264.762,Z 701.008,A -85,B 0,C 180,E1 -18923.34,E2 -18923.34} C_VEL
LIN {X 0,Y 262.318,Z 712.888,A -85,B 0,C 180,E1 -18924.893,E2 -18924.893} C_VEL
LIN {X 0,Y 259.697,Z 723.899,A -85,B 0,C 180,E1 -18926.746,E2 -18926.746} C_VEL
LIN {X 0,Y 256.928,Z 734.027,A -85,B 0,C 180,E1 -18928.922,E2 -18928.922} C_VEL
LIN {X 0,Y 254.533,Z 742.19,A -85,B 0,C 180,E1 -18931.14,E2 -18931.14} C_VEL
LIN {X 0,Y 252.504,Z 748.76,A -85,B 0,C 180,E1 -18933.39,E2 -18933.39} C_VEL
LIN {X 0,Y 250.486,Z 754.939,A -85,B 0,C 180,E1 -18936.1,E2 -18936.1} C_VEL
LIN {X 0,Y 249.224,Z 758.874,A -85,B 0,C 180,E1 -18938.343,E2 -18938.343} C_VEL
LIN {X 0,Y 248.262,Z 761.927,A -85,B 0,C 180,E1 -18940.624,E2 -18940.624} C_VEL
LIN {X 0,Y 247.515,Z 764.148,A -85,B 0,C 180,E1 -18942.957,E2 -18942.957} C_VEL
LIN {X 0,Y 246.989,Z 765.515,A -85,B 0,C 180,E1 -18945.345,E2 -18945.345} C_VEL
LIN {X 0,Y 246.661,Z 766.009,A -85,B 0,C 180,E1 -18947.799,E2 -18947.799} C_VEL
LIN {X 0,Y 246.536,Z 765.576,A -85,B 0,C 180,E1 -18950.324,E2 -18950.324} C_VEL
LIN {X 0,Y 246.688,Z 763.875,A -85,B 0,C 180,E1 -18953.257,E2 -18953.257} C_VEL
LIN {X 0,Y 247.223,Z 760.375,A -85,B 0,C 180,E1 -18956.479,E2 -18956.479} C_VEL
LIN {X 0,Y 247.861,Z 755.836,A -85,B 0,C 180,E1 -18959.314,E2 -18959.314} C_VEL
LIN {X 0,Y 248.733,Z 750.634,A -85,B 0,C 180,E1 -18961.756,E2 -18961.756} C_VEL
LIN {X 0,Y 249.879,Z 744.134,A -85,B 0,C 180,E1 -18964.159,E2 -18964.159} C_VEL
LIN {X 0,Y 251.32,Z 736.119,A -85,B 0,C 180,E1 -18966.519,E2 -18966.519} C_VEL
LIN {X 0,Y 252.899,Z 727.302,A -85,B 0,C 180,E1 -18968.611,E2 -18968.611} C_VEL
LIN {X 0,Y 254.44,Z 718.122,A -85,B 0,C 180,E1 -18970.382,E2 -18970.382} C_VEL
LIN {X 0,Y 256.148,Z 707.499,A -85,B 0,C 180,E1 -18972.023,E2 -18972.023} C_VEL
LIN {X 0,Y 257.653,Z 695.987,A -85,B 0,C 180,E1 -18973.434,E2 -18973.434} C_VEL
LIN {X 0,Y 259.046,Z 683.949,A -85,B 0,C 180,E1 -18974.564,E2 -18974.564} C_VEL
LIN {X 0,Y 260.144,Z 670.691,A -85,B 0,C 180,E1 -18975.457,E2 -18975.457} C_VEL
LIN {X 0,Y 260.949,Z 657.443,A -85,B 0,C 180,E1 -18976.024,E2 -18976.024} C_VEL
LIN {X 0,Y 263.336,Z 592.382,A -85,B 0,C 180,E1 -18977.943,E2 -18977.943} C_VEL
LIN {X 0,Y 260.4,Z 583.259,A -85,B 0,C 180,E1 -18978.518,E2 -18978.518} C_VEL
LIN {X 0,Y 252.718,Z 562.861,A -85,B 0,C 180,E1 -18979.977,E2 -18979.977} C_VEL
LIN {X 0,Y 249.718,Z 555.094,A -85,B 0,C 180,E1 -18980.579,E2 -18980.579} C_VEL
LIN {X 0,Y 249.446,Z 553.414,A -85,B 0,C 180,E1 -18981.386,E2 -18981.386} C_VEL
